LIN {X 0,Y 347.835,Z 893.328,A -85,B 0,C 180,E1 -23554.002,E2 -23554.002} C_VEL
LIN {X 0,Y 356.996,Z 872.801,A -85,B 0,C 180,E1 -23555.35,E2 -23555.35} C_VEL
LIN {X 0,Y 365.708,Z 850.209,A -85,B 0,C 180,E1 -23556.534,E2 -23556.534} C_VEL
LIN {X 0,Y 372.164,Z 830.904,A -85,B 0,C 180,E1 -23557.35,E2 -23557.35} C_VEL
LIN {X 0,Y 378.965,Z 806.777,A -85,B 0,C 180,E1 -23558.164,E2 -23558.164} C_VEL
LIN {X 0,Y 383.904,Z 784.469,A -85,B 0,C 180,E1 -23558.738,E2 -23558.738} C_VEL
LIN {X 0,Y 388.031,Z 759.695,A -85,B 0,C 180,E1 -23559.245,E2 -23559.245} C_VEL
LIN {X 0,Y 393.244,Z 706.009,A -85,B 0,C 180,E1 -23560.109,E2 -23560.109} C_VEL
LIN {X 0,Y 405.179,Z 577.067,A -85,B 0,C 180,E1 -23562.107,E2 -23562.107} C_VEL
LIN {X 0,Y 400.868,Z 567.631,A -85,B 0,C 180,E1 -23564.706,E2 -23564.706} C_VEL
LIN {X 0,Y 397.081,Z 560.851,A -85,B 0,C 180,E1 -23567.345,E2 -23567.345} C_VEL
LIN {X 0,Y 394.785,Z 556.79,A -85,B 0,C 180,E1 -23569.271,E2 -23569.271} C_VEL
LIN {X 0,Y 393.127,Z 553.806,A -85,B 0,C 180,E1 -23570.927,E2 -23570.927} C_VEL
LIN {X 0,Y 390.899,Z 549.726,A -85,B 0,C 180,E1 -23573.833,E2 -23573.833} C_VEL
LIN {X 0,Y 389.05,Z 545.081,A -85,B 0,C 180,E1 -23580.295,E2 -23580.295} C_VEL
LIN {X 0,Y 391.195,Z 550.264,A -85,B 0,C 180,E1 -23587.047,E2 -23587.047} C_VEL
LIN {X 0,Y 393.909,Z 555.208,A -85,B 0,C 180,E1 -23590.309,E2 -23590.309} C_VEL
LIN {X 0,Y 396.663,Z 560.048,A -85,B 0,C 180,E1 -23592.742,E2 -23592.742} C_VEL
LIN {X 0,Y 400.307,Z 566.598,A -85,B 0,C 180,E1 -23595.353,E2 -23595.353} C_VEL
LIN {X 0,Y 405.195,Z 575.818,A -85,B 0,C 180,E1 -23598.251,E2 -23598.251} C_VEL
LIN {X 0,Y 389.01,Z 748.36,A -85,B 0,C 180,E1 -23600.94,E2 -23600.94} C_VEL
LIN {X 0,Y 384.925,Z 774.814,A -85,B 0,C 180,E1 -23601.482,E2 -23601.482} C_VEL
LIN {X 0,Y 380.503,Z 795.662,A -85,B 0,C 180,E1 -23602.045,E2 -23602.045} C_VEL
LIN {X 0,Y 373.946,Z 820.335,A -85,B 0,C 180,E1 -23602.905,E2 -23602.905} C_VEL
LIN {X 0,Y 367.245,Z 840.974,A -85,B 0,C 180,E1 -23603.82,E2 -23603.82} C_VEL
LIN {X 0,Y 358.727,Z 863.66,A -85,B 0,C 180,E1 -23605.058,E2 -23605.058} C_VEL
LIN {X 0,Y 349.576,Z 884.374,A -85,B 0,C 180,E1 -23606.457,E2 -23606.457} C_VEL
LIN {X 0,Y 339.93,Z 904.027,A -85,B 0,C 180,E1 -23608.063,E2 -23608.063} C_VEL
LIN {X 0,Y 329.108,Z 923.521,A -85,B 0,C 180,E1 -23610.017,E2 -23610.017} C_VEL
LIN {X 0,Y 319.02,Z 940.165,A -85,B 0,C 180,E1 -23612.025,E2 -23612.025} C_VEL
LIN {X 0,Y 306.526,Z 958.98,A -85,B 0,C 180,E1 -23614.81,E2 -23614.81} C_VEL
LIN {X 0,Y 296.049,Z 973.609,A -85,B 0,C 180,E1 -23617.468,E2 -23617.468} C_VEL
LIN {X 0,Y 283.786,Z 989.665,A -85,B 0,C 180,E1 -23621.062,E2 -23621.062} C_VEL
LIN {X 0,Y 273.785,Z 1002.093,A -85,B 0,C 180,E1 -23624.524,E2 -23624.524} C_VEL
LIN {X 0,Y 263.22,Z 1014.833,A -85,B 0,C 180,E1 -23628.916,E2 -23628.916} C_VEL
LIN {X 0,Y 254.603,Z 1024.994,A -85,B 0,C 180,E1 -23633.349,E2 -23633.349} C_VEL
LIN {X 0,Y 246.801,Z 1034.427,A -85,B 0,C 180,E1 -23638.491,E2 -23638.491} C_VEL
LIN {X 0,Y 240.758,Z 1041.973,A -85,B 0,C 180,E1 -23643.882,E2 -23643.882} C_VEL
LIN {X 0,Y 236.318,Z 1048.28,A -85,B 0,C 180,E1 -23649.699,E2 -23649.699} C_VEL
LIN {X 0,Y 233.696,Z 1052.582,A -85,B 0,C 180,E1 -23655.378,E2 -23655.378} C_VEL
LIN {X 0,Y 232.543,Z 1055.206,A -85,B 0,C 180,E1 -23660.347,E2 -23660.347} C_VEL
LIN {X 0,Y 232.083,Z 1056.918,A -85,B 0,C 180,E1 -23665.8,E2 -23665.8} C_VEL
LIN {X 0,Y 232.025,Z 1057.239,A -85,B 0,C 180,E1 -23670.988,E2 -23670.988} C_VEL
LIN {X 0,Y 232.144,Z 1056.542,A -85,B 0,C 180,E1 -23675.751,E2 -23675.751} C_VEL
LIN {X 0,Y 232.638,Z 1054.939,A -85,B 0,C 180,E1 -23680.4,E2 -23680.4} C_VEL
LIN {X 0,Y 234.023,Z 1052.049,A -85,B 0,C 180,E1 -23685.615,E2 -23685.615} C_VEL
LIN {X 0,Y 237.201,Z 1046.942,A -85,B 0,C 180,E1 -23691.775,E2 -23691.775} C_VEL
LIN {X 0,Y 241.377,Z 1041.246,A -85,B 0,C 180,E1 -23696.842,E2 -23696.842} C_VEL
LIN {X 0,Y 248.254,Z 1032.711,A -85,B 0,C 180,E1 -23702.664,E2 -23702.664} C_VEL
LIN {X 0,Y 255.637,Z 1023.876,A -85,B 0,C 180,E1 -23707.32,E2 -23707.32} C_VEL
LIN {X 0,Y 265.345,Z 1012.444,A -85,B 0,C 180,E1 -23712.125,E2 -23712.125} C_VEL
LIN {X 0,Y 275.066,Z 1000.672,A -85,B 0,C 180,E1 -23716.034,E2 -23716.034} C_VEL
LIN {X 0,Y 285.965,Z 987.176,A -85,B 0,C 180,E1 -23719.694,E2 -23719.694} C_VEL
LIN {X 0,Y 297.122,Z 972.362,A -85,B 0,C 180,E1 -23722.898,E2 -23722.898} C_VEL
LIN {X 0,Y 307.93,Z 957.247,A -85,B 0,C 180,E1 -23725.597,E2 -23725.597} C_VEL
LIN {X 0,Y 319.887,Z 939.064,A -85,B 0,C 180,E1 -23728.234,E2 -23728.234} C_VEL
LIN {X 0,Y 330.019,Z 922.313,A -85,B 0,C 180,E1 -23730.231,E2 -23730.231} C_VEL
LIN {X 0,Y 341.605,Z 901.102,A -85,B 0,C 180,E1 -23732.305,E2 -23732.305} C_VEL
LIN {X 0,Y 350.412,Z 883.055,A -85,B 0,C 180,E1 -23733.75,E2 -23733.75} C_VEL
LIN {X 0,Y 359.976,Z 861.087,A -85,B 0,C 180,E1 -23735.201,E2 -23735.201} C_VEL
LIN {X 0,Y 367.879,Z 839.801,A -85,B 0,C 180,E1 -23736.343,E2 -23736.343} C_VEL
LIN {X 0,Y 375.388,Z 816.305,A -85,B 0,C 180,E1 -23737.361,E2 -23737.361} C_VEL
LIN {X 0,Y 381.309,Z 793.174,A -85,B 0,C 180,E1 -23738.135,E2 -23738.135} C_VEL
LIN {X 0,Y 386.229,Z 769.254,A -85,B 0,C 180,E1 -23738.756,E2 -23738.756} C_VEL
LIN {X 0,Y 389.656,Z 744.741,A -85,B 0,C 180,E1 -23739.225,E2 -23739.225} C_VEL
LIN {X 0,Y 405.413,Z 575.97,A -85,B 0,C 180,E1 -23741.857,E2 -23741.857} C_VEL
LIN {X 0,Y 400.628,Z 566.958,A -85,B 0,C 180,E1 -23744.696,E2 -23744.696} C_VEL
LIN {X 0,Y 397.121,Z 560.633,A -85,B 0,C 180,E1 -23747.199,E2 -23747.199} C_VEL
LIN {X 0,Y 395.089,Z 557.156,A -85,B 0,C 180,E1 -23748.911,E2 -23748.911} C_VEL
LIN {X 0,Y 393.763,Z 554.568,A -85,B 0,C 180,E1 -23750.233,E2 -23750.233} C_VEL
LIN {X 0,Y 392.838,Z 553.605,A -85,B 0,C 180,E1 -23751.18,E2 -23751.18} C_VEL
LIN {X 0,Y 391.337,Z 554.58,A -85,B 0,C 180,E1 -23752.628,E2 -23752.628} C_VEL
LIN {X 0,Y 389.554,Z 556.788,A -85,B 0,C 180,E1 -23754.674,E2 -23754.674} C_VEL
LIN {X 0,Y 389.136,Z 556.727,A -85,B 0,C 180,E1 -23755.421,E2 -23755.421} C_VEL
LIN {X 0,Y 388.33,Z 553.902,A -85,B 0,C 180,E1 -23760,E2 -23760} C_VEL
LIN {X 0,Y 390.299,Z 558.224,A -85,B 0,C 180,E1 -23766.325,E2 -23766.325} C_VEL
LIN {X 0,Y 392.89,Z 563.078,A -85,B 0,C 180,E1 -23769.596,E2 -23769.596} C_VEL
LIN {X 0,Y 395.281,Z 567.502,A -85,B 0,C 180,E1 -23771.823,E2 -23771.823} C_VEL
LIN {X 0,Y 398.829,Z 573.955,A -85,B 0,C 180,E1 -23774.482,E2 -23774.482} C_VEL
LIN {X 0,Y 401.266,Z 579.253,A -85,B 0,C 180,E1 -23776.094,E2 -23776.094} C_VEL
LIN {X 0,Y 402.503,Z 582.459,A -85,B 0,C 180,E1 -23776.88,E2 -23776.88} C_VEL
LIN {X 0,Y 385.936,Z 755.658,A -85,B 0,C 180,E1 -23779.56,E2 -23779.56} C_VEL
LIN {X 0,Y 381.709,Z 782.23,A -85,B 0,C 180,E1 -23780.078,E2 -23780.078} C_VEL
LIN {X 0,Y 376.982,Z 803.644,A -85,B 0,C 180,E1 -23780.604,E2 -23780.604} C_VEL
LIN {X 0,Y 369.986,Z 828.756,A -85,B 0,C 180,E1 -23781.406,E2 -23781.406} C_VEL
LIN {X 0,Y 363.401,Z 848.284,A -85,B 0,C 180,E1 -23782.199,E2 -23782.199} C_VEL
LIN {X 0,Y 354.645,Z 870.927,A -85,B 0,C 180,E1 -23783.34,E2 -23783.34} C_VEL
LIN {X 0,Y 345.022,Z 892.161,A -85,B 0,C 180,E1 -23784.696,E2 -23784.696} C_VEL
LIN {X 0,Y 334.593,Z 912.794,A -85,B 0,C 180,E1 -23786.296,E2 -23786.296} C_VEL
LIN {X 0,Y 323.349,Z 932.438,A -85,B 0,C 180,E1 -23788.2,E2 -23788.2} C_VEL
LIN {X 0,Y 312.514,Z 949.839,A -85,B 0,C 180,E1 -23790.246,E2 -23790.246} C_VEL
LIN {X 0,Y 300.014,Z 968.143,A -85,B 0,C 180,E1 -23792.905,E2 -23792.905} C_VEL
LIN {X 0,Y 288.971,Z 983.211,A -85,B 0,C 180,E1 -23795.596,E2 -23795.596} C_VEL
LIN {X 0,Y 276.215,Z 999.555,A -85,B 0,C 180,E1 -23799.224,E2 -23799.224} C_VEL
LIN {X 0,Y 265.688,Z 1012.399,A -85,B 0,C 180,E1 -23802.789,E2 -23802.789} C_VEL
LIN {X 0,Y 253.914,Z 1026.348,A -85,B 0,C 180,E1 -23807.671,E2 -23807.671} C_VEL
LIN {X 0,Y 245.528,Z 1036.235,A -85,B 0,C 180,E1 -23812.053,E2 -23812.053} C_VEL
LIN {X 0,Y 236.986,Z 1046.589,A -85,B 0,C 180,E1 -23817.885,E2 -23817.885} C_VEL
LIN {X 0,Y 231.559,Z 1053.665,A -85,B 0,C 180,E1 -23823.038,E2 -23823.038} C_VEL
LIN {X 0,Y 227.283,Z 1060.146,A -85,B 0,C 180,E1 -23829.124,E2 -23829.124} C_VEL
LIN {X 0,Y 225.031,Z 1064.472,A -85,B 0,C 180,E1 -23834.802,E2 -23834.802} C_VEL
LIN {X 0,Y 224.137,Z 1067.258,A -85,B 0,C 180,E1 -23839.98,E2 -23839.98} C_VEL
LIN {X 0,Y 223.98,Z 1069.011,A -85,B 0,C 180,E1 -23845.391,E2 -23845.391} C_VEL
LIN {X 0,Y 224.019,Z 1069.447,A -85,B 0,C 180,E1 -23850.511,E2 -23850.511} C_VEL
LIN {X 0,Y 223.982,Z 1068.773,A -85,B 0,C 180,E1 -23855.43,E2 -23855.43} C_VEL
LIN {X 0,Y 224.163,Z 1067.118,A -85,B 0,C 180,E1 -23860.278,E2 -23860.278} C_VEL
LIN {X 0,Y 225.102,Z 1064.276,A -85,B 0,C 180,E1 -23865.457,E2 -23865.457} C_VEL
LIN {X 0,Y 227.71,Z 1059.396,A -85,B 0,C 180,E1 -23871.644,E2 -23871.644} C_VEL
LIN {X 0,Y 232.007,Z 1052.984,A -85,B 0,C 180,E1 -23877.461,E2 -23877.461} C_VEL
LIN {X 0,Y 238.204,Z 1045.073,A -85,B 0,C 180,E1 -23883.072,E2 -23883.072} C_VEL
LIN {X 0,Y 246.352,Z 1035.142,A -85,B 0,C 180,E1 -23888.432,E2 -23888.432} C_VEL
LIN {X 0,Y 255.749,Z 1024.154,A -85,B 0,C 180,E1 -23893.172,E2 -23893.172} C_VEL
LIN {X 0,Y 266.497,Z 1011.26,A -85,B 0,C 180,E1 -23897.518,E2 -23897.518} C_VEL
LIN {X 0,Y 277.466,Z 997.863,A -85,B 0,C 180,E1 -23901.168,E2 -23901.168} C_VEL
LIN {X 0,Y 289.588,Z 982.165,A -85,B 0,C 180,E1 -23904.573,E2 -23904.573} C_VEL
LIN {X 0,Y 300.731,Z 966.912,A -85,B 0,C 180,E1 -23907.266,E2 -23907.266} C_VEL
LIN {X 0,Y 313.412,Z 948.132,A -85,B 0,C 180,E1 -23909.941,E2 -23909.941} C_VEL
LIN {X 0,Y 323.697,Z 931.53,A -85,B 0,C 180,E1 -23911.872,E2 -23911.872} C_VEL
LIN {X 0,Y 335.331,Z 910.95,A -85,B 0,C 180,E1 -23913.834,E2 -23913.834} C_VEL
LIN {X 0,Y 344.999,Z 891.755,A -85,B 0,C 180,E1 -23915.312,E2 -23915.312} C_VEL
LIN {X 0,Y 354.893,Z 869.78,A -85,B 0,C 180,E1 -23916.705,E2 -23916.705} C_VEL
LIN {X 0,Y 363.376,Z 847.717,A -85,B 0,C 180,E1 -23917.81,E2 -23917.81} C_VEL
LIN {X 0,Y 370.996,Z 824.871,A -85,B 0,C 180,E1 -23918.724,E2 -23918.724} C_VEL
LIN {X 0,Y 377.303,Z 801.317,A -85,B 0,C 180,E1 -23919.444,E2 -23919.444} C_VEL
LIN {X 0,Y 382.253,Z 778.324,A -85,B 0,C 180,E1 -23919.995,E2 -23919.995} C_VEL
LIN {X 0,Y 385.966,Z 753.258,A -85,B 0,C 180,E1 -23920.467,E2 -23920.467} C_VEL
LIN {X 0,Y 402.254,Z 581.98,A -85,B 0,C 180,E1 -23923.133,E2 -23923.133} C_VEL
LIN {X 0,Y 399.045,Z 574.683,A -85,B 0,C 180,E1 -23925.192,E2 -23925.192} C_VEL
LIN {X 0,Y 395.538,Z 568.236,A -85,B 0,C 180,E1 -23927.74,E2 -23927.74} C_VEL
LIN {X 0,Y 393.361,Z 564.263,A -85,B 0,C 180,E1 -23929.646,E2 -23929.646} C_VEL
LIN {X 0,Y 391.874,Z 561.512,A -85,B 0,C 180,E1 -23931.194,E2 -23931.194} C_VEL
LIN {X 0,Y 389.826,Z 557.61,A -85,B 0,C 180,E1 -23933.963,E2 -23933.963} C_VEL
LIN {X 0,Y 388.07,Z 553.065,A -85,B 0,C 180,E1 -23940.295,E2 -23940.295} C_VEL
LIN {X 0,Y 390.11,Z 558.197,A -85,B 0,C 180,E1 -23946.919,E2 -23946.919} C_VEL
LIN {X 0,Y 392.633,Z 562.902,A -85,B 0,C 180,E1 -23950.046,E2 -23950.046} C_VEL
LIN {X 0,Y 395.301,Z 567.74,A -85,B 0,C 180,E1 -23952.483,E2 -23952.483} C_VEL
LIN {X 0,Y 398.867,Z 574.383,A -85,B 0,C 180,E1 -23955.112,E2 -23955.112} C_VEL
LIN {X 0,Y 402.28,Z 581.103,A -85,B 0,C 180,E1 -23957.247,E2 -23957.247} C_VEL
LIN {X 0,Y 386.223,Z 748.596,A -85,B 0,C 180,E1 -23959.831,E2 -23959.831} C_VEL
LIN {X 0,Y 382.065,Z 775.041,A -85,B 0,C 180,E1 -23960.365,E2 -23960.365} C_VEL
LIN {X 0,Y 377.539,Z 796.006,A -85,B 0,C 180,E1 -23960.92,E2 -23960.92} C_VEL
LIN {X 0,Y 370.894,Z 820.557,A -85,B 0,C 180,E1 -23961.762,E2 -23961.762} C_VEL
LIN {X 0,Y 364.072,Z 841.195,A -85,B 0,C 180,E1 -23962.663,E2 -23962.663} C_VEL
LIN {X 0,Y 355.785,Z 862.969,A -85,B 0,C 180,E1 -23963.826,E2 -23963.826} C_VEL
LIN {X 0,Y 346.372,Z 883.931,A -85,B 0,C 180,E1 -23965.212,E2 -23965.212} C_VEL
LIN {X 0,Y 337.315,Z 902.058,A -85,B 0,C 180,E1 -23966.655,E2 -23966.655} C_VEL
LIN {X 0,Y 325.851,Z 922.533,A -85,B 0,C 180,E1 -23968.646,E2 -23968.646} C_VEL
LIN {X 0,Y 315.826,Z 938.734,A -85,B 0,C 180,E1 -23970.556,E2 -23970.556} C_VEL
LIN {X 0,Y 303.797,Z 956.658,A -85,B 0,C 180,E1 -23973.118,E2 -23973.118} C_VEL
LIN {X 0,Y 292.406,Z 972.156,A -85,B 0,C 180,E1 -23975.863,E2 -23975.863} C_VEL
LIN {X 0,Y 280.816,Z 987.093,A -85,B 0,C 180,E1 -23979.084,E2 -23979.084} C_VEL
LIN {X 0,Y 269.51,Z 1000.635,A -85,B 0,C 180,E1 -23982.761,E2 -23982.761} C_VEL
LIN {X 0,Y 259.43,Z 1012.375,A -85,B 0,C 180,E1 -23986.683,E2 -23986.683} C_VEL
LIN {X 0,Y 249.261,Z 1023.861,A -85,B 0,C 180,E1 -23991.555,E2 -23991.555} C_VEL
LIN {X 0,Y 241.36,Z 1032.85,A -85,B 0,C 180,E1 -23996.377,E2 -23996.377} C_VEL
LIN {X 0,Y 234.159,Z 1041.303,A -85,B 0,C 180,E1 -24002.261,E2 -24002.261} C_VEL
LIN {X 0,Y 229.684,Z 1047.025,A -85,B 0,C 180,E1 -24007.475,E2 -24007.475} C_VEL
LIN {X 0,Y 226.24,Z 1052.18,A -85,B 0,C 180,E1 -24013.833,E2 -24013.833} C_VEL
LIN {X 0,Y 224.717,Z 1055.093,A -85,B 0,C 180,E1 -24019.229,E2 -24019.229} C_VEL
LIN {X 0,Y 224.158,Z 1056.737,A -85,B 0,C 180,E1 -24024.115,E2 -24024.115} C_VEL
LIN {X 0,Y 224.027,Z 1057.44,A -85,B 0,C 180,E1 -24028.977,E2 -24028.977} C_VEL
LIN {X 0,Y 224.09,Z 1057.164,A -85,B 0,C 180,E1 -24034.351,E2 -24034.351} C_VEL
LIN {X 0,Y 224.582,Z 1055.484,A -85,B 0,C 180,E1 -24040,E2 -24040} C_VEL
LIN {X 0,Y 225.839,Z 1052.874,A -85,B 0,C 180,E1 -24045.162,E2 -24045.162} C_VEL
LIN {X 0,Y 228.796,Z 1048.397,A -85,B 0,C 180,E1 -24051.268,E2 -24051.268} C_VEL
LIN {X 0,Y 233.361,Z 1042.353,A -85,B 0,C 180,E1 -24057.013,E2 -24057.013} C_VEL
LIN {X 0,Y 239.429,Z 1035.18,A -85,B 0,C 180,E1 -24062.313,E2 -24062.313} C_VEL
LIN {X 0,Y 247.945,Z 1025.449,A -85,B 0,C 180,E1 -24067.805,E2 -24067.805} C_VEL
LIN {X 0,Y 256.495,Z 1015.819,A -85,B 0,C 180,E1 -24072.106,E2 -24072.106} C_VEL
LIN {X 0,Y 267.838,Z 1002.771,A -85,B 0,C 180,E1 -24076.717,E2 -24076.717} C_VEL
LIN {X 0,Y 278.342,Z 990.221,A -85,B 0,C 180,E1 -24080.25,E2 -24080.25} C_VEL
LIN {X 0,Y 291,Z 974.252,A -85,B 0,C 180,E1 -24083.85,E2 -24083.85} C_VEL
LIN {X 0,Y 301.322,Z 960.303,A -85,B 0,C 180,E1 -24086.398,E2 -24086.398} C_VEL
LIN {X 0,Y 313.583,Z 942.582,A -85,B 0,C 180,E1 -24089.063,E2 -24089.063} C_VEL
LIN {X 0,Y 324.607,Z 924.941,A -85,B 0,C 180,E1 -24091.205,E2 -24091.205} C_VEL
LIN {X 0,Y 335.672,Z 905.662,A -85,B 0,C 180,E1 -24093.144,E2 -24093.144} C_VEL
LIN {X 0,Y 345.903,Z 885.378,A -85,B 0,C 180,E1 -24094.794,E2 -24094.794} C_VEL
LIN {X 0,Y 355.023,Z 865.225,A -85,B 0,C 180,E1 -24096.143,E2 -24096.143} C_VEL
LIN {X 0,Y 363.927,Z 842.261,A -85,B 0,C 180,E1 -24097.393,E2 -24097.393} C_VEL
LIN {X 0,Y 370.753,Z 821.765,A -85,B 0,C 180,E1 -24098.293,E2 -24098.293} C_VEL
LIN {X 0,Y 377.704,Z 796.339,A -85,B 0,C 180,E1 -24099.173,E2 -24099.173} C_VEL
LIN {X 0,Y 382.228,Z 775.446,A -85,B 0,C 180,E1 -24099.729,E2 -24099.729} C_VEL
LIN {X 0,Y 386.349,Z 749.637,A -85,B 0,C 180,E1 -24100.255,E2 -24100.255} C_VEL
LIN {X 0,Y 395.791,Z 651.868,A -85,B 0,C 180,E1 -24101.779,E2 -24101.779} C_VEL
LIN {X 0,Y 402.488,Z 581.077,A -85,B 0,C 180,E1 -24102.879,E2 -24102.879} C_VEL
LIN {X 0,Y 398.217,Z 572.864,A -85,B 0,C 180,E1 -24105.606,E2 -24105.606} C_VEL
LIN {X 0,Y 394.679,Z 566.202,A -85,B 0,C 180,E1 -24108.381,E2 -24108.381} C_VEL
LIN {X 0,Y 391.99,Z 561.546,A -85,B 0,C 180,E1 -24111.048,E2 -24111.048} C_VEL
LIN {X 0,Y 390.009,Z 557.709,A -85,B 0,C 180,E1 -24113.818,E2 -24113.818} C_VEL
LIN {X 0,Y 389.136,Z 556.727,A -85,B 0,C 180,E1 -24115.421,E2 -24115.421} C_VEL
LIN {X 0,Y 388.526,Z 556.957,A -85,B 0,C 180,E1 -24116.725,E2 -24116.725} C_VEL
LIN {X 0,Y 387.342,Z 562.179,A -85,B 0,C 180,E1 -24120.541,E2 -24120.541} C_VEL
LIN {X 0,Y 387.342,Z 562.238,A -85,B 0,C 180,E1 -24120.624,E2 -24120.624} C_VEL
LIN {X 0,Y 389.22,Z 566.147,A -85,B 0,C 180,E1 -24126.194,E2 -24126.194} C_VEL
LIN {X 0,Y 391.624,Z 570.769,A -85,B 0,C 180,E1 -24129.33,E2 -24129.33} C_VEL
LIN {X 0,Y 393.943,Z 575.21,A -85,B 0,C 180,E1 -24131.567,E2 -24131.567} C_VEL
LIN {X 0,Y 397.303,Z 581.526,A -85,B 0,C 180,E1 -24134.167,E2 -24134.167} C_VEL
LIN {X 0,Y 399.766,Z 587.148,A -85,B 0,C 180,E1 -24135.852,E2 -24135.852} C_VEL
LIN {X 0,Y 383.322,Z 755.464,A -85,B 0,C 180,E1 -24138.429,E2 -24138.429} C_VEL
LIN {X 0,Y 379.026,Z 782.029,A -85,B 0,C 180,E1 -24138.937,E2 -24138.937} C_VEL
LIN {X 0,Y 374.227,Z 803.44,A -85,B 0,C 180,E1 -24139.451,E2 -24139.451} C_VEL
LIN {X 0,Y 367.087,Z 828.651,A -85,B 0,C 180,E1 -24140.239,E2 -24140.239} C_VEL
LIN {X 0,Y 360.013,Z 849.21,A -85,B 0,C 180,E1 -24141.061,E2 -24141.061} C_VEL
LIN {X 0,Y 350.975,Z 871.908,A -85,B 0,C 180,E1 -24142.197,E2 -24142.197} C_VEL
LIN {X 0,Y 341.309,Z 892.765,A -85,B 0,C 180,E1 -24143.515,E2 -24143.515} C_VEL
LIN {X 0,Y 330.675,Z 913.297,A -85,B 0,C 180,E1 -24145.092,E2 -24145.092} C_VEL
LIN {X 0,Y 319.19,Z 932.836,A -85,B 0,C 180,E1 -24146.973,E2 -24146.973} C_VEL
LIN {X 0,Y 307.378,Z 951.301,A -85,B 0,C 180,E1 -24149.141,E2 -24149.141} C_VEL
LIN {X 0,Y 294.996,Z 968.776,A -85,B 0,C 180,E1 -24151.705,E2 -24151.705} C_VEL
LIN {X 0,Y 283.598,Z 983.847,A -85,B 0,C 180,E1 -24154.409,E2 -24154.409} C_VEL
LIN {X 0,Y 271.059,Z 999.336,A -85,B 0,C 180,E1 -24157.869,E2 -24157.869} C_VEL
LIN {X 0,Y 260.126,Z 1012.18,A -85,B 0,C 180,E1 -24161.448,E2 -24161.448} C_VEL
LIN {X 0,Y 247.845,Z 1026.128,A -85,B 0,C 180,E1 -24166.38,E2 -24166.38} C_VEL
LIN {X 0,Y 239.039,Z 1036.015,A -85,B 0,C 180,E1 -24170.83,E2 -24170.83} C_VEL
LIN {X 0,Y 230.013,Z 1046.369,A -85,B 0,C 180,E1 -24176.788,E2 -24176.788} C_VEL
LIN {X 0,Y 224.23,Z 1053.446,A -85,B 0,C 180,E1 -24182.081,E2 -24182.081} C_VEL
LIN {X 0,Y 219.627,Z 1059.927,A -85,B 0,C 180,E1 -24188.36,E2 -24188.36} C_VEL
LIN {X 0,Y 217.168,Z 1064.255,A -85,B 0,C 180,E1 -24194.237,E2 -24194.237} C_VEL
LIN {X 0,Y 216.172,Z 1067.042,A -85,B 0,C 180,E1 -24199.607,E2 -24199.607} C_VEL
LIN {X 0,Y 215.982,Z 1068.797,A -85,B 0,C 180,E1 -24205.22,E2 -24205.22} C_VEL
LIN {X 0,Y 216.024,Z 1069.256,A -85,B 0,C 180,E1 -24210.265,E2 -24210.265} C_VEL
LIN {X 0,Y 215.984,Z 1068.585,A -85,B 0,C 180,E1 -24215.532,E2 -24215.532} C_VEL
LIN {X 0,Y 216.199,Z 1066.902,A -85,B 0,C 180,E1 -24220.661,E2 -24220.661} C_VEL
LIN {X 0,Y 217.247,Z 1064.058,A -85,B 0,C 180,E1 -24226.03,E2 -24226.03} C_VEL
LIN {X 0,Y 220.088,Z 1059.176,A -85,B 0,C 180,E1 -24232.434,E2 -24232.434} C_VEL
LIN {X 0,Y 224.708,Z 1052.763,A -85,B 0,C 180,E1 -24238.432,E2 -24238.432} C_VEL
LIN {X 0,Y 231.308,Z 1044.85,A -85,B 0,C 180,E1 -24244.191,E2 -24244.191} C_VEL
LIN {X 0,Y 239.846,Z 1034.987,A -85,B 0,C 180,E1 -24249.631,E2 -24249.631} C_VEL
LIN {X 0,Y 249.763,Z 1023.931,A -85,B 0,C 180,E1 -24254.474,E2 -24254.474} C_VEL
LIN {X 0,Y 260.66,Z 1011.398,A -85,B 0,C 180,E1 -24258.751,E2 -24258.751} C_VEL
LIN {X 0,Y 271.815,Z 998.273,A -85,B 0,C 180,E1 -24262.364,E2 -24262.364} C_VEL
LIN {X 0,Y 284.232,Z 982.796,A -85,B 0,C 180,E1 -24265.761,E2 -24265.761} C_VEL
LIN {X 0,Y 295.01,Z 968.512,A -85,B 0,C 180,E1 -24268.308,E2 -24268.308} C_VEL
LIN {X 0,Y 307.72,Z 950.474,A -85,B 0,C 180,E1 -24270.935,E2 -24270.935} C_VEL
LIN {X 0,Y 319.168,Z 932.533,A -85,B 0,C 180,E1 -24273.034,E2 -24273.034} C_VEL
LIN {X 0,Y 330.653,Z 912.94,A -85,B 0,C 180,E1 -24274.915,E2 -24274.915} C_VEL
LIN {X 0,Y 341.285,Z 892.349,A -85,B 0,C 180,E1 -24276.494,E2 -24276.494} C_VEL
LIN {X 0,Y 350.952,Z 871.453,A -85,B 0,C 180,E1 -24277.812,E2 -24277.812} C_VEL
LIN {X 0,Y 359.988,Z 848.629,A -85,B 0,C 180,E1 -24278.949,E2 -24278.949} C_VEL
LIN {X 0,Y 367.517,Z 826.592,A -85,B 0,C 180,E1 -24279.822,E2 -24279.822} C_VEL
LIN {X 0,Y 374.231,Z 802.425,A -85,B 0,C 180,E1 -24280.561,E2 -24280.561} C_VEL
LIN {X 0,Y 379.017,Z 780.857,A -85,B 0,C 180,E1 -24281.074,E2 -24281.074} C_VEL
LIN {X 0,Y 383.196,Z 754.379,A -85,B 0,C 180,E1 -24281.576,E2 -24281.576} C_VEL
LIN {X 0,Y 399.508,Z 586.924,A -85,B 0,C 180,E1 -24284.148,E2 -24284.148} C_VEL
LIN {X 0,Y 397.002,Z 581.207,A -85,B 0,C 180,E1 -24285.859,E2 -24285.859} C_VEL
LIN {X 0,Y 392.968,Z 573.447,A -85,B 0,C 180,E1 -24289.073,E2 -24289.073} C_VEL
LIN {X 0,Y 390.63,Z 569.218,A -85,B 0,C 180,E1 -24291.462,E2 -24291.462} C_VEL
LIN {X 0,Y 388.661,Z 565.407,A -85,B 0,C 180,E1 -24294.242,E2 -24294.242} C_VEL
LIN {X 0,Y 387.09,Z 561.048,A -85,B 0,C 180,E1 -24300.296,E2 -24300.296} C_VEL
LIN {X 0,Y 388.986,Z 566.008,A -85,B 0,C 180,E1 -24306.717,E2 -24306.717} C_VEL
LIN {X 0,Y 391.365,Z 570.596,A -85,B 0,C 180,E1 -24309.782,E2 -24309.782} C_VEL
LIN {X 0,Y 393.964,Z 575.461,A -85,B 0,C 180,E1 -24312.235,E2 -24312.235} C_VEL
LIN {X 0,Y 397.588,Z 582.47,A -85,B 0,C 180,E1 -24314.976,E2 -24314.976} C_VEL
LIN {X 0,Y 399.474,Z 586.526,A -85,B 0,C 180,E1 -24316.23,E2 -24316.23} C_VEL
LIN {X 0,Y 383.559,Z 749.024,A -85,B 0,C 180,E1 -24318.71,E2 -24318.71} C_VEL
LIN {X 0,Y 379.331,Z 775.378,A -85,B 0,C 180,E1 -24319.234,E2 -24319.234} C_VEL
LIN {X 0,Y 374.723,Z 796.351,A -85,B 0,C 180,E1 -24319.779,E2 -24319.779} C_VEL
LIN {X 0,Y 367.993,Z 820.78,A -85,B 0,C 180,E1 -24320.601,E2 -24320.601} C_VEL
LIN {X 0,Y 361.05,Z 841.417,A -85,B 0,C 180,E1 -24321.485,E2 -24321.485} C_VEL
LIN {X 0,Y 352.476,Z 863.496,A -85,B 0,C 180,E1 -24322.646,E2 -24322.646} C_VEL
LIN {X 0,Y 342.687,Z 884.816,A -85,B 0,C 180,E1 -24324.039,E2 -24324.039} C_VEL
LIN {X 0,Y 332.617,Z 904.469,A -85,B 0,C 180,E1 -24325.6,E2 -24325.6} C_VEL
LIN {X 0,Y 321.293,Z 923.962,A -85,B 0,C 180,E1 -24327.509,E2 -24327.509} C_VEL
LIN {X 0,Y 311.049,Z 940.057,A -85,B 0,C 180,E1 -24329.408,E2 -24329.408} C_VEL
LIN {X 0,Y 297.716,Z 959.149,A -85,B 0,C 180,E1 -24332.183,E2 -24332.183} C_VEL
LIN {X 0,Y 287.041,Z 973.214,A -85,B 0,C 180,E1 -24334.705,E2 -24334.705} C_VEL
LIN {X 0,Y 274.506,Z 988.721,A -85,B 0,C 180,E1 -24338.115,E2 -24338.115} C_VEL
LIN {X 0,Y 263.508,Z 1001.419,A -85,B 0,C 180,E1 -24341.624,E2 -24341.624} C_VEL
LIN {X 0,Y 252.527,Z 1013.727,A -85,B 0,C 180,E1 -24345.823,E2 -24345.823} C_VEL
LIN {X 0,Y 242.451,Z 1024.533,A -85,B 0,C 180,E1 -24350.572,E2 -24350.572} C_VEL
LIN {X 0,Y 233.983,Z 1033.733,A -85,B 0,C 180,E1 -24355.662,E2 -24355.662} C_VEL
LIN {X 0,Y 226.67,Z 1041.82,A -85,B 0,C 180,E1 -24361.549,E2 -24361.549} C_VEL
LIN {X 0,Y 221.785,Z 1047.741,A -85,B 0,C 180,E1 -24367.188,E2 -24367.188} C_VEL
LIN {X 0,Y 218.236,Z 1052.707,A -85,B 0,C 180,E1 -24373.771,E2 -24373.771} C_VEL
LIN {X 0,Y 216.74,Z 1055.418,A -85,B 0,C 180,E1 -24379.097,E2 -24379.097} C_VEL
LIN {X 0,Y 216.159,Z 1057.016,A -85,B 0,C 180,E1 -24384.159,E2 -24384.159} C_VEL
LIN {X 0,Y 216.026,Z 1057.698,A -85,B 0,C 180,E1 -24389.47,E2 -24389.47} C_VEL
LIN {X 0,Y 216.119,Z 1057.25,A -85,B 0,C 180,E1 -24395.043,E2 -24395.043} C_VEL
LIN {X 0,Y 216.678,Z 1055.589,A -85,B 0,C 180,E1 -24400.637,E2 -24400.637} C_VEL
LIN {X 0,Y 218.106,Z 1052.946,A -85,B 0,C 180,E1 -24405.966,E2 -24405.966} C_VEL
LIN {X 0,Y 221.379,Z 1048.37,A -85,B 0,C 180,E1 -24412.297,E2 -24412.297} C_VEL
LIN {X 0,Y 226.34,Z 1042.275,A -85,B 0,C 180,E1 -24418.209,E2 -24418.209} C_VEL
LIN {X 0,Y 233.203,Z 1034.705,A -85,B 0,C 180,E1 -24423.876,E2 -24423.876} C_VEL
LIN {X 0,Y 241.918,Z 1025.215,A -85,B 0,C 180,E1 -24429.226,E2 -24429.226} C_VEL
LIN {X 0,Y 251.911,Z 1014.515,A -85,B 0,C 180,E1 -24433.997,E2 -24433.997} C_VEL
LIN {X 0,Y 263.083,Z 1002.063,A -85,B 0,C 180,E1 -24438.308,E2 -24438.308} C_VEL
LIN {X 0,Y 274.364,Z 989.069,A -85,B 0,C 180,E1 -24441.924,E2 -24441.924} C_VEL
LIN {X 0,Y 286.897,Z 973.63,A -85,B 0,C 180,E1 -24445.336,E2 -24445.336} C_VEL
LIN {X 0,Y 297.568,Z 959.6,A -85,B 0,C 180,E1 -24447.863,E2 -24447.863} C_VEL
LIN {X 0,Y 310.545,Z 941.144,A -85,B 0,C 180,E1 -24450.57,E2 -24450.57} C_VEL
LIN {X 0,Y 321.369,Z 924.187,A -85,B 0,C 180,E1 -24452.582,E2 -24452.582} C_VEL
LIN {X 0,Y 332.855,Z 904.447,A -85,B 0,C 180,E1 -24454.515,E2 -24454.515} C_VEL
LIN {X 0,Y 342.542,Z 885.589,A -85,B 0,C 180,E1 -24456.016,E2 -24456.016} C_VEL
LIN {X 0,Y 351.695,Z 865.757,A -85,B 0,C 180,E1 -24457.325,E2 -24457.325} C_VEL
LIN {X 0,Y 360.58,Z 843.387,A -85,B 0,C 180,E1 -24458.528,E2 -24458.528} C_VEL
LIN {X 0,Y 367.448,Z 823.252,A -85,B 0,C 180,E1 -24459.404,E2 -24459.404} C_VEL
LIN {X 0,Y 374.39,Z 798.814,A -85,B 0,C 180,E1 -24460.25,E2 -24460.25} C_VEL
LIN {X 0,Y 379.189,Z 777.337,A -85,B 0,C 180,E1 -24460.824,E2 -24460.824} C_VEL
LIN {X 0,Y 383.356,Z 752.93,A -85,B 0,C 180,E1 -24461.328,E2 -24461.328} C_VEL
LIN {X 0,Y 388.692,Z 700.563,A -85,B 0,C 180,E1 -24462.149,E2 -24462.149} C_VEL
LIN {X 0,Y 399.734,Z 586.426,A -85,B 0,C 180,E1 -24463.88,E2 -24463.88} C_VEL
LIN {X 0,Y 395.755,Z 578.597,A -85,B 0,C 180,E1 -24466.633,E2 -24466.633} C_VEL
LIN {X 0,Y 392.799,Z 573.044,A -85,B 0,C 180,E1 -24469.142,E2 -24469.142} C_VEL
LIN {X 0,Y 390.881,Z 569.436,A -85,B 0,C 180,E1 -24471.171,E2 -24471.171} C_VEL
LIN {X 0,Y 388.853,Z 565.503,A -85,B 0,C 180,E1 -24474.096,E2 -24474.096} C_VEL
LIN {X 0,Y 387.353,Z 561.858,A -85,B 0,C 180,E1 -24480,E2 -24480} C_VEL
LIN {X 0,Y 387.342,Z 562.238,A -85,B 0,C 180,E1 -24480.624,E2 -24480.624} C_VEL
LIN {X 0,Y 387.305,Z 563.992,A -85,B 0,C 180,E1 -24481.743,E2 -24481.743} C_VEL
LIN {X 0,Y 387.45,Z 572.167,A -85,B 0,C 180,E1 -24484.643,E2 -24484.643} C_VEL
LIN {X 0,Y 387.889,Z 573.488,A -85,B 0,C 180,E1 -24485.604,E2 -24485.604} C_VEL
LIN {X 0,Y 390.367,Z 578.459,A -85,B 0,C 180,E1 -24489.063,E2 -24489.063} C_VEL
LIN {X 0,Y 392.702,Z 583.09,A -85,B 0,C 180,E1 -24491.388,E2 -24491.388} C_VEL
LIN {X 0,Y 395.886,Z 589.303,A -85,B 0,C 180,E1 -24493.92,E2 -24493.92} C_VEL
LIN {X 0,Y 397.105,Z 592.406,A -85,B 0,C 180,E1 -24494.819,E2 -24494.819} C_VEL
LIN {X 0,Y 380.859,Z 755.271,A -85,B 0,C 180,E1 -24497.283,E2 -24497.283} C_VEL
LIN {X 0,Y 376.49,Z 781.862,A -85,B 0,C 180,E1 -24497.782,E2 -24497.782} C_VEL
LIN {X 0,Y 371.6,Z 803.345,A -85,B 0,C 180,E1 -24498.285,E2 -24498.285} C_VEL
LIN {X 0,Y 364.41,Z 828.344,A -85,B 0,C 180,E1 -24499.046,E2 -24499.046} C_VEL
LIN {X 0,Y 357.188,Z 849.001,A -85,B 0,C 180,E1 -24499.851,E2 -24499.851} C_VEL
LIN {X 0,Y 347.996,Z 871.698,A -85,B 0,C 180,E1 -24500.962,E2 -24500.962} C_VEL
LIN {X 0,Y 338.151,Z 892.553,A -85,B 0,C 180,E1 -24502.253,E2 -24502.253} C_VEL
LIN {X 0,Y 327.304,Z 913.083,A -85,B 0,C 180,E1 -24503.801,E2 -24503.801} C_VEL
LIN {X 0,Y 315.567,Z 932.621,A -85,B 0,C 180,E1 -24505.65,E2 -24505.65} C_VEL
LIN {X 0,Y 303.643,Z 950.828,A -85,B 0,C 180,E1 -24507.758,E2 -24507.758} C_VEL
LIN {X 0,Y 290.758,Z 968.559,A -85,B 0,C 180,E1 -24510.326,E2 -24510.326} C_VEL
LIN {X 0,Y 279.021,Z 983.629,A -85,B 0,C 180,E1 -24513.012,E2 -24513.012} C_VEL
LIN {X 0,Y 265.44,Z 999.826,A -85,B 0,C 180,E1 -24516.644,E2 -24516.644} C_VEL
LIN {X 0,Y 254.149,Z 1012.603,A -85,B 0,C 180,E1 -24520.248,E2 -24520.248} C_VEL
LIN {X 0,Y 241.908,Z 1025.908,A -85,B 0,C 180,E1 -24525.024,E2 -24525.024} C_VEL
LIN {X 0,Y 232.664,Z 1035.795,A -85,B 0,C 180,E1 -24529.539,E2 -24529.539} C_VEL
LIN {X 0,Y 223.13,Z 1046.149,A -85,B 0,C 180,E1 -24535.623,E2 -24535.623} C_VEL
LIN {X 0,Y 216.861,Z 1053.354,A -85,B 0,C 180,E1 -24541.169,E2 -24541.169} C_VEL
LIN {X 0,Y 211.85,Z 1059.921,A -85,B 0,C 180,E1 -24547.816,E2 -24547.816} C_VEL
LIN {X 0,Y 209.24,Z 1064.203,A -85,B 0,C 180,E1 -24553.909,E2 -24553.909} C_VEL
LIN {X 0,Y 208.181,Z 1066.945,A -85,B 0,C 180,E1 -24559.484,E2 -24559.484} C_VEL
LIN {X 0,Y 207.983,Z 1068.651,A -85,B 0,C 180,E1 -24565.312,E2 -24565.312} C_VEL
LIN {X 0,Y 208.025,Z 1069.02,A -85,B 0,C 180,E1 -24570.551,E2 -24570.551} C_VEL
LIN {X 0,Y 207.986,Z 1068.358,A -85,B 0,C 180,E1 -24575.794,E2 -24575.794} C_VEL
LIN {X 0,Y 208.24,Z 1066.685,A -85,B 0,C 180,E1 -24581.073,E2 -24581.073} C_VEL
LIN {X 0,Y 209.41,Z 1063.84,A -85,B 0,C 180,E1 -24586.648,E2 -24586.648} C_VEL
LIN {X 0,Y 212.505,Z 1058.955,A -85,B 0,C 180,E1 -24593.281,E2 -24593.281} C_VEL
LIN {X 0,Y 217.472,Z 1052.541,A -85,B 0,C 180,E1 -24599.469,E2 -24599.469} C_VEL
LIN {X 0,Y 224.583,Z 1044.541,A -85,B 0,C 180,E1 -24605.437,E2 -24605.437} C_VEL
LIN {X 0,Y 233.517,Z 1034.764,A -85,B 0,C 180,E1 -24610.929,E2 -24610.929} C_VEL
LIN {X 0,Y 243.911,Z 1023.708,A -85,B 0,C 180,E1 -24615.84,E2 -24615.84} C_VEL
LIN {X 0,Y 255.273,Z 1011.175,A -85,B 0,C 180,E1 -24620.149,E2 -24620.149} C_VEL
LIN {X 0,Y 266.673,Z 998.245,A -85,B 0,C 180,E1 -24623.72,E2 -24623.72} C_VEL
LIN {X 0,Y 279.676,Z 982.573,A -85,B 0,C 180,E1 -24627.157,E2 -24627.157} C_VEL
LIN {X 0,Y 290.739,Z 968.335,A -85,B 0,C 180,E1 -24629.68,E2 -24629.68} C_VEL
LIN {X 0,Y 303.822,Z 950.252,A -85,B 0,C 180,E1 -24632.287,E2 -24632.287} C_VEL
LIN {X 0,Y 315.546,Z 932.311,A -85,B 0,C 180,E1 -24634.357,E2 -24634.357} C_VEL
LIN {X 0,Y 327.418,Z 912.47,A -85,B 0,C 180,E1 -24636.227,E2 -24636.227} C_VEL
LIN {X 0,Y 338.165,Z 892.055,A -85,B 0,C 180,E1 -24637.761,E2 -24637.761} C_VEL
LIN {X 0,Y 347.974,Z 871.231,A -85,B 0,C 180,E1 -24639.047,E2 -24639.047} C_VEL
LIN {X 0,Y 357.165,Z 848.407,A -85,B 0,C 180,E1 -24640.158,E2 -24640.158} C_VEL
LIN {X 0,Y 364.814,Z 826.369,A -85,B 0,C 180,E1 -24641.011,E2 -24641.011} C_VEL
LIN {X 0,Y 371.652,Z 802.115,A -85,B 0,C 180,E1 -24641.732,E2 -24641.732} C_VEL
LIN {X 0,Y 376.535,Z 780.405,A -85,B 0,C 180,E1 -24642.236,E2 -24642.236} C_VEL
LIN {X 0,Y 380.746,Z 754.035,A -85,B 0,C 180,E1 -24642.725,E2 -24642.725} C_VEL
LIN {X 0,Y 396.863,Z 591.973,A -85,B 0,C 180,E1 -24645.183,E2 -24645.183} C_VEL
LIN {X 0,Y 394.714,Z 587.291,A -85,B 0,C 180,E1 -24646.747,E2 -24646.747} C_VEL
LIN {X 0,Y 391.346,Z 580.637,A -85,B 0,C 180,E1 -24649.623,E2 -24649.623} C_VEL
LIN {X 0,Y 389.395,Z 576.922,A -85,B 0,C 180,E1 -24651.732,E2 -24651.732} C_VEL
LIN {X 0,Y 387.595,Z 573.29,A -85,B 0,C 180,E1 -24654.374,E2 -24654.374} C_VEL
LIN {X 0,Y 386.11,Z 569.031,A -85,B 0,C 180,E1 -24660.297,E2 -24660.297} C_VEL
LIN {X 0,Y 387.907,Z 573.936,A -85,B 0,C 180,E1 -24666.587,E2 -24666.587} C_VEL
LIN {X 0,Y 390.17,Z 578.433,A -85,B 0,C 180,E1 -24669.589,E2 -24669.589} C_VEL
LIN {X 0,Y 392.627,Z 583.166,A -85,B 0,C 180,E1 -24671.979,E2 -24671.979} C_VEL
LIN {X 0,Y 396.416,Z 590.741,A -85,B 0,C 180,E1 -24674.909,E2 -24674.909} C_VEL
LIN {X 0,Y 396.815,Z 591.739,A -85,B 0,C 180,E1 -24675.195,E2 -24675.195} C_VEL
LIN {X 0,Y 381.068,Z 749.259,A -85,B 0,C 180,E1 -24677.57,E2 -24677.57} C_VEL
LIN {X 0,Y 376.791,Z 775.495,A -85,B 0,C 180,E1 -24678.081,E2 -24678.081} C_VEL
LIN {X 0,Y 372.087,Z 796.576,A -85,B 0,C 180,E1 -24678.617,E2 -24678.617} C_VEL
LIN {X 0,Y 365.245,Z 821.003,A -85,B 0,C 180,E1 -24679.422,E2 -24679.422} C_VEL
LIN {X 0,Y 358.184,Z 841.639,A -85,B 0,C 180,E1 -24680.288,E2 -24680.288} C_VEL
LIN {X 0,Y 349.587,Z 863.409,A -85,B 0,C 180,E1 -24681.41,E2 -24681.41} C_VEL
LIN {X 0,Y 339.88,Z 884.23,A -85,B 0,C 180,E1 -24682.738,E2 -24682.738} C_VEL
LIN {X 0,Y 329.976,Z 903.23,A -85,B 0,C 180,E1 -24684.205,E2 -24684.205} C_VEL
LIN {X 0,Y 318.005,Z 923.578,A -85,B 0,C 180,E1 -24686.145,E2 -24686.145} C_VEL
LIN {X 0,Y 307.133,Z 940.278,A -85,B 0,C 180,E1 -24688.085,E2 -24688.085} C_VEL
LIN {X 0,Y 293.449,Z 959.37,A -85,B 0,C 180,E1 -24690.834,E2 -24690.834} C_VEL
LIN {X 0,Y 282.463,Z 973.435,A -85,B 0,C 180,E1 -24693.341,E2 -24693.341} C_VEL
LIN {X 0,Y 269.526,Z 988.942,A -85,B 0,C 180,E1 -24696.744,E2 -24696.744} C_VEL
LIN {X 0,Y 257.82,Z 1001.978,A -85,B 0,C 180,E1 -24700.366,E2 -24700.366} C_VEL
LIN {X 0,Y 246.186,Z 1014.482,A -85,B 0,C 180,E1 -24704.703,E2 -24704.703} C_VEL
LIN {X 0,Y 235.717,Z 1025.205,A -85,B 0,C 180,E1 -24709.533,E2 -24709.533} C_VEL
LIN {X 0,Y 226.523,Z 1034.738,A -85,B 0,C 180,E1 -24714.983,E2 -24714.983} C_VEL
LIN {X 0,Y 219.219,Z 1042.336,A -85,B 0,C 180,E1 -24720.788,E2 -24720.788} C_VEL
LIN {X 0,Y 213.892,Z 1048.456,A -85,B 0,C 180,E1 -24726.879,E2 -24726.879} C_VEL
LIN {X 0,Y 210.338,Z 1053.079,A -85,B 0,C 180,E1 -24733.428,E2 -24733.428} C_VEL
LIN {X 0,Y 208.734,Z 1055.807,A -85,B 0,C 180,E1 -24739.115,E2 -24739.115} C_VEL
LIN {X 0,Y 208.122,Z 1057.494,A -85,B 0,C 180,E1 -24745.039,E2 -24745.039} C_VEL
LIN {X 0,Y 208.032,Z 1057.901,A -85,B 0,C 180,E1 -24750.826,E2 -24750.826} C_VEL
LIN {X 0,Y 208.178,Z 1057.246,A -85,B 0,C 180,E1 -24756.153,E2 -24756.153} C_VEL
LIN {X 0,Y 208.861,Z 1055.584,A -85,B 0,C 180,E1 -24761.6,E2 -24761.6} C_VEL
LIN {X 0,Y 210.764,Z 1052.544,A -85,B 0,C 180,E1 -24767.676,E2 -24767.676} C_VEL
LIN {X 0,Y 214.617,Z 1047.594,A -85,B 0,C 180,E1 -24774.204,E2 -24774.204} C_VEL
LIN {X 0,Y 219.7,Z 1041.9,A -85,B 0,C 180,E1 -24779.741,E2 -24779.741} C_VEL
LIN {X 0,Y 227.512,Z 1033.763,A -85,B 0,C 180,E1 -24785.769,E2 -24785.769} C_VEL
LIN {X 0,Y 236.046,Z 1024.982,A -85,B 0,C 180,E1 -24790.719,E2 -24790.719} C_VEL
LIN {X 0,Y 246.573,Z 1014.22,A -85,B 0,C 180,E1 -24795.537,E2 -24795.537} C_VEL
LIN {X 0,Y 257.996,Z 1001.951,A -85,B 0,C 180,E1 -24799.774,E2 -24799.774} C_VEL
LIN {X 0,Y 270.014,Z 988.593,A -85,B 0,C 180,E1 -24803.473,E2 -24803.473} C_VEL
LIN {X 0,Y 282.338,Z 973.827,A -85,B 0,C 180,E1 -24806.706,E2 -24806.706} C_VEL
LIN {X 0,Y 293.634,Z 959.387,A -85,B 0,C 180,E1 -24809.284,E2 -24809.284} C_VEL
LIN {X 0,Y 307.397,Z 940.201,A -85,B 0,C 180,E1 -24812.042,E2 -24812.042} C_VEL
LIN {X 0,Y 318.244,Z 923.554,A -85,B 0,C 180,E1 -24813.973,E2 -24813.973} C_VEL
LIN {X 0,Y 330.228,Z 903.198,A -85,B 0,C 180,E1 -24815.91,E2 -24815.91} C_VEL
LIN {X 0,Y 339.801,Z 884.872,A -85,B 0,C 180,E1 -24817.326,E2 -24817.326} C_VEL
LIN {X 0,Y 349.45,Z 864.256,A -85,B 0,C 180,E1 -24818.648,E2 -24818.648} C_VEL
LIN {X 0,Y 358.345,Z 841.877,A -85,B 0,C 180,E1 -24819.806,E2 -24819.806} C_VEL
LIN {X 0,Y 365.534,Z 820.898,A -85,B 0,C 180,E1 -24820.686,E2 -24820.686} C_VEL
LIN {X 0,Y 372.434,Z 796.204,A -85,B 0,C 180,E1 -24821.497,E2 -24821.497} C_VEL
LIN {X 0,Y 377.163,Z 774.936,A -85,B 0,C 180,E1 -24822.035,E2 -24822.035} C_VEL
LIN {X 0,Y 381.454,Z 748.203,A -85,B 0,C 180,E1 -24822.55,E2 -24822.55} C_VEL
LIN {X 0,Y 397.072,Z 591.697,A -85,B 0,C 180,E1 -24824.917,E2 -24824.917} C_VEL
LIN {X 0,Y 393.162,Z 583.892,A -85,B 0,C 180,E1 -24827.888,E2 -24827.888} C_VEL
LIN {X 0,Y 390.926,Z 579.693,A -85,B 0,C 180,E1 -24829.984,E2 -24829.984} C_VEL
LIN {X 0,Y 389.526,Z 576.964,A -85,B 0,C 180,E1 -24831.586,E2 -24831.586} C_VEL
LIN {X 0,Y 387.791,Z 573.386,A -85,B 0,C 180,E1 -24834.229,E2 -24834.229} C_VEL
LIN {X 0,Y 386.376,Z 569.819,A -85,B 0,C 180,E1 -24840,E2 -24840} C_VEL
LIN {X 0,Y 387.889,Z 573.488,A -85,B 0,C 180,E1 -24845.604,E2 -24845.604} C_VEL
LIN {X 0,Y 388.403,Z 575.002,A -85,B 0,C 180,E1 -24846.551,E2 -24846.551} C_VEL
LIN {X 0,Y 388.923,Z 579.017,A -85,B 0,C 180,E1 -24847.721,E2 -24847.721} C_VEL
LIN {X 0,Y 390.018,Z 587.241,A -85,B 0,C 180,E1 -24849.713,E2 -24849.713} C_VEL
LIN {X 0,Y 390.552,Z 588.948,A -85,B 0,C 180,E1 -24850.323,E2 -24850.323} C_VEL
LIN {X 0,Y 394.102,Z 596.247,A -85,B 0,C 180,E1 -24853.386,E2 -24853.386} C_VEL
LIN {X 0,Y 394.581,Z 597.586,A -85,B 0,C 180,E1 -24853.771,E2 -24853.771} C_VEL
LIN {X 0,Y 378.539,Z 755.173,A -85,B 0,C 180,E1 -24856.123,E2 -24856.123} C_VEL
LIN {X 0,Y 374.103,Z 781.719,A -85,B 0,C 180,E1 -24856.612,E2 -24856.612} C_VEL
LIN {X 0,Y 369.102,Z 803.358,A -85,B 0,C 180,E1 -24857.106,E2 -24857.106} C_VEL
LIN {X 0,Y 361.86,Z 828.136,A -85,B 0,C 180,E1 -24857.839,E2 -24857.839} C_VEL
LIN {X 0,Y 354.527,Z 848.792,A -85,B 0,C 180,E1 -24858.623,E2 -24858.623} C_VEL
LIN {X 0,Y 344.94,Z 872.005,A -85,B 0,C 180,E1 -24859.735,E2 -24859.735} C_VEL
LIN {X 0,Y 335.16,Z 892.342,A -85,B 0,C 180,E1 -24860.968,E2 -24860.968} C_VEL
LIN {X 0,Y 323.984,Z 913.071,A -85,B 0,C 180,E1 -24862.501,E2 -24862.501} C_VEL
LIN {X 0,Y 312.121,Z 932.4,A -85,B 0,C 180,E1 -24864.297,E2 -24864.297} C_VEL
LIN {X 0,Y 300.119,Z 950.311,A -85,B 0,C 180,E1 -24866.335,E2 -24866.335} C_VEL
LIN {X 0,Y 287.425,Z 967.409,A -85,B 0,C 180,E1 -24868.758,E2 -24868.758} C_VEL
LIN {X 0,Y 276.006,Z 981.706,A -85,B 0,C 180,E1 -24871.244,E2 -24871.244} C_VEL
LIN {X 0,Y 262.534,Z 997.482,A -85,B 0,C 180,E1 -24874.648,E2 -24874.648} C_VEL
LIN {X 0,Y 250.659,Z 1010.456,A -85,B 0,C 180,E1 -24878.201,E2 -24878.201} C_VEL
LIN {X 0,Y 238.75,Z 1023.065,A -85,B 0,C 180,E1 -24882.516,E2 -24882.516} C_VEL
LIN {X 0,Y 227.577,Z 1034.384,A -85,B 0,C 180,E1 -24887.573,E2 -24887.573} C_VEL
LIN {X 0,Y 218.173,Z 1044.101,A -85,B 0,C 180,E1 -24893.103,E2 -24893.103} C_VEL
LIN {X 0,Y 210.399,Z 1052.289,A -85,B 0,C 180,E1 -24899.337,E2 -24899.337} C_VEL
LIN {X 0,Y 205.156,Z 1058.527,A -85,B 0,C 180,E1 -24905.526,E2 -24905.526} C_VEL
LIN {X 0,Y 201.694,Z 1063.49,A -85,B 0,C 180,E1 -24912.398,E2 -24912.398} C_VEL
LIN {X 0,Y 200.326,Z 1066.375,A -85,B 0,C 180,E1 -24918.191,E2 -24918.191} C_VEL
LIN {X 0,Y 199.986,Z 1068.086,A -85,B 0,C 180,E1 -24923.685,E2 -24923.685} C_VEL
LIN {X 0,Y 200.023,Z 1068.765,A -85,B 0,C 180,E1 -24928.854,E2 -24928.854} C_VEL
LIN {X 0,Y 199.989,Z 1068.52,A -85,B 0,C 180,E1 -24934.014,E2 -24934.014} C_VEL
LIN {X 0,Y 200.136,Z 1067.058,A -85,B 0,C 180,E1 -24940.07,E2 -24940.07} C_VEL
LIN {X 0,Y 201.318,Z 1064.117,A -85,B 0,C 180,E1 -24946.445,E2 -24946.445} C_VEL
LIN {X 0,Y 203.921,Z 1060.085,A -85,B 0,C 180,E1 -24952.486,E2 -24952.486} C_VEL
LIN {X 0,Y 209.497,Z 1053.25,A -85,B 0,C 180,E1 -24959.76,E2 -24959.76} C_VEL
LIN {X 0,Y 215.984,Z 1046.21,A -85,B 0,C 180,E1 -24965.358,E2 -24965.358} C_VEL
LIN {X 0,Y 225.996,Z 1035.903,A -85,B 0,C 180,E1 -24971.606,E2 -24971.606} C_VEL
LIN {X 0,Y 235.813,Z 1025.866,A -85,B 0,C 180,E1 -24976.279,E2 -24976.279} C_VEL
LIN {X 0,Y 248.694,Z 1012.42,A -85,B 0,C 180,E1 -24981.155,E2 -24981.155} C_VEL
LIN {X 0,Y 259.931,Z 1000.148,A -85,B 0,C 180,E1 -24984.638,E2 -24984.638} C_VEL
LIN {X 0,Y 273.219,Z 984.911,A -85,B 0,C 180,E1 -24988.107,E2 -24988.107} C_VEL
LIN {X 0,Y 285.947,Z 969.046,A -85,B 0,C 180,E1 -24990.949,E2 -24990.949} C_VEL
LIN {X 0,Y 298.958,Z 951.688,A -85,B 0,C 180,E1 -24993.466,E2 -24993.466} C_VEL
LIN {X 0,Y 311.308,Z 933.314,A -85,B 0,C 180,E1 -24995.584,E2 -24995.584} C_VEL
LIN {X 0,Y 322.554,Z 915.042,A -85,B 0,C 180,E1 -24997.308,E2 -24997.308} C_VEL
LIN {X 0,Y 334.31,Z 893.536,A -85,B 0,C 180,E1 -24998.933,E2 -24998.933} C_VEL
LIN {X 0,Y 343.472,Z 874.624,A -85,B 0,C 180,E1 -25000.1,E2 -25000.1} C_VEL
LIN {X 0,Y 353.652,Z 850.453,A -85,B 0,C 180,E1 -25001.29,E2 -25001.29} C_VEL
LIN {X 0,Y 361.017,Z 829.883,A -85,B 0,C 180,E1 -25002.084,E2 -25002.084} C_VEL
LIN {X 0,Y 368.253,Z 805.713,A -85,B 0,C 180,E1 -25002.82,E2 -25002.82} C_VEL
LIN {X 0,Y 373.482,Z 783.429,A -85,B 0,C 180,E1 -25003.34,E2 -25003.34} C_VEL
LIN {X 0,Y 377.853,Z 758.646,A -85,B 0,C 180,E1 -25003.808,E2 -25003.808} C_VEL
LIN {X 0,Y 383.618,Z 703.877,A -85,B 0,C 180,E1 -25004.647,E2 -25004.647} C_VEL
LIN {X 0,Y 394.322,Z 597.081,A -85,B 0,C 180,E1 -25006.244,E2 -25006.244} C_VEL
LIN {X 0,Y 391.102,Z 590.543,A -85,B 0,C 180,E1 -25008.871,E2 -25008.871} C_VEL
LIN {X 0,Y 388.54,Z 585.184,A -85,B 0,C 180,E1 -25011.565,E2 -25011.565} C_VEL
LIN {X 0,Y 386.531,Z 581.173,A -85,B 0,C 180,E1 -25014.508,E2 -25014.508} C_VEL
LIN {X 0,Y 385.129,Z 577.015,A -85,B 0,C 180,E1 -25020.298,E2 -25020.298} C_VEL
LIN {X 0,Y 386.79,Z 581.745,A -85,B 0,C 180,E1 -25026.382,E2 -25026.382} C_VEL
LIN {X 0,Y 388.979,Z 586.268,A -85,B 0,C 180,E1 -25029.394,E2 -25029.394} C_VEL
LIN {X 0,Y 391.379,Z 591.028,A -85,B 0,C 180,E1 -25031.793,E2 -25031.793} C_VEL
LIN {X 0,Y 394.277,Z 597.06,A -85,B 0,C 180,E1 -25034.149,E2 -25034.149} C_VEL
LIN {X 0,Y 378.729,Z 749.495,A -85,B 0,C 180,E1 -25036.416,E2 -25036.416} C_VEL
LIN {X 0,Y 374.384,Z 775.722,A -85,B 0,C 180,E1 -25036.916,E2 -25036.916} C_VEL
LIN {X 0,Y 369.605,Z 796.802,A -85,B 0,C 180,E1 -25037.439,E2 -25037.439} C_VEL
LIN {X 0,Y 362.655,Z 821.225,A -85,B 0,C 180,E1 -25038.226,E2 -25038.226} C_VEL
LIN {X 0,Y 355.477,Z 841.861,A -85,B 0,C 180,E1 -25039.073,E2 -25039.073} C_VEL
LIN {X 0,Y 346.586,Z 863.948,A -85,B 0,C 180,E1 -25040.188,E2 -25040.188} C_VEL
LIN {X 0,Y 336.841,Z 884.451,A -85,B 0,C 180,E1 -25041.472,E2 -25041.472} C_VEL
LIN {X 0,Y 327.251,Z 902.513,A -85,B 0,C 180,E1 -25042.833,E2 -25042.833} C_VEL
LIN {X 0,Y 314.901,Z 923.195,A -85,B 0,C 180,E1 -25044.753,E2 -25044.753} C_VEL
LIN {X 0,Y 303.764,Z 939.948,A -85,B 0,C 180,E1 -25046.66,E2 -25046.66} C_VEL
LIN {X 0,Y 289.97,Z 958.803,A -85,B 0,C 180,E1 -25049.318,E2 -25049.318} C_VEL
LIN {X 0,Y 278.05,Z 973.656,A -85,B 0,C 180,E1 -25051.933,E2 -25051.933} C_VEL
LIN {X 0,Y 264.705,Z 989.163,A -85,B 0,C 180,E1 -25055.323,E2 -25055.323} C_VEL
LIN {X 0,Y 252.903,Z 1001.861,A -85,B 0,C 180,E1 -25058.843,E2 -25058.843} C_VEL
LIN {X 0,Y 241.009,Z 1014.169,A -85,B 0,C 180,E1 -25063.099,E2 -25063.099} C_VEL
LIN {X 0,Y 229.738,Z 1025.219,A -85,B 0,C 180,E1 -25068.095,E2 -25068.095} C_VEL
LIN {X 0,Y 220.222,Z 1034.572,A -85,B 0,C 180,E1 -25073.503,E2 -25073.503} C_VEL
LIN {X 0,Y 212.286,Z 1042.367,A -85,B 0,C 180,E1 -25079.537,E2 -25079.537} C_VEL
LIN {X 0,Y 206.814,Z 1048.179,A -85,B 0,C 180,E1 -25085.431,E2 -25085.431} C_VEL
LIN {X 0,Y 202.684,Z 1053.142,A -85,B 0,C 180,E1 -25092.487,E2 -25092.487} C_VEL
LIN {X 0,Y 200.906,Z 1055.85,A -85,B 0,C 180,E1 -25098.226,E2 -25098.226} C_VEL
LIN {X 0,Y 200.175,Z 1057.511,A -85,B 0,C 180,E1 -25103.979,E2 -25103.979} C_VEL
LIN {X 0,Y 200.038,Z 1058.168,A -85,B 0,C 180,E1 -25110,E2 -25110} C_VEL
LIN {X 0,Y 200.173,Z 1057.546,A -85,B 0,C 180,E1 -25116.022,E2 -25116.022} C_VEL
LIN {X 0,Y 200.891,Z 1055.909,A -85,B 0,C 180,E1 -25121.775,E2 -25121.775} C_VEL
LIN {X 0,Y 202.775,Z 1053.07,A -85,B 0,C 180,E1 -25127.802,E2 -25127.802} C_VEL
LIN {X 0,Y 207.185,Z 1047.812,A -85,B 0,C 180,E1 -25135.132,E2 -25135.132} C_VEL
LIN {X 0,Y 212.615,Z 1042.118,A -85,B 0,C 180,E1 -25140.838,E2 -25140.838} C_VEL
LIN {X 0,Y 220.894,Z 1033.981,A -85,B 0,C 180,E1 -25147.016,E2 -25147.016} C_VEL
LIN {X 0,Y 229.875,Z 1025.2,A -85,B 0,C 180,E1 -25152.056,E2 -25152.056} C_VEL
LIN {X 0,Y 240.885,Z 1014.438,A -85,B 0,C 180,E1 -25156.934,E2 -25156.934} C_VEL
LIN {X 0,Y 252.771,Z 1002.168,A -85,B 0,C 180,E1 -25161.195,E2 -25161.195} C_VEL
LIN {X 0,Y 265.216,Z 988.81,A -85,B 0,C 180,E1 -25164.896,E2 -25164.896} C_VEL
LIN {X 0,Y 277.914,Z 974.062,A -85,B 0,C 180,E1 -25168.113,E2 -25168.113} C_VEL
LIN {X 0,Y 289.211,Z 960.03,A -85,B 0,C 180,E1 -25170.603,E2 -25170.603} C_VEL
LIN {X 0,Y 302.875,Z 941.571,A -85,B 0,C 180,E1 -25173.254,E2 -25173.254} C_VEL
LIN {X 0,Y 313.987,Z 924.976,A -85,B 0,C 180,E1 -25175.174,E2 -25175.174} C_VEL
LIN {X 0,Y 325.814,Z 905.6,A -85,B 0,C 180,E1 -25177.024,E2 -25177.024} C_VEL
LIN {X 0,Y 336.301,Z 886.009,A -85,B 0,C 180,E1 -25178.53,E2 -25178.53} C_VEL
LIN {X 0,Y 345.763,Z 866.258,A -85,B 0,C 180,E1 -25179.785,E2 -25179.785} C_VEL
LIN {X 0,Y 355.065,Z 843.648,A -85,B 0,C 180,E1 -25180.952,E2 -25180.952} C_VEL
LIN {X 0,Y 362.37,Z 822.872,A -85,B 0,C 180,E1 -25181.815,E2 -25181.815} C_VEL
LIN {X 0,Y 369.808,Z 797.056,A -85,B 0,C 180,E1 -25182.656,E2 -25182.656} C_VEL
LIN {X 0,Y 374.609,Z 775.917,A -85,B 0,C 180,E1 -25183.182,E2 -25183.182} C_VEL
LIN {X 0,Y 378.962,Z 749.785,A -85,B 0,C 180,E1 -25183.681,E2 -25183.681} C_VEL
LIN {X 0,Y 391.906,Z 623.162,A -85,B 0,C 180,E1 -25185.571,E2 -25185.571} C_VEL
LIN {X 0,Y 394.526,Z 597.237,A -85,B 0,C 180,E1 -25185.956,E2 -25185.956} C_VEL
LIN {X 0,Y 391.344,Z 590.649,A -85,B 0,C 180,E1 -25188.579,E2 -25188.579} C_VEL
LIN {X 0,Y 388.546,Z 585.036,A -85,B 0,C 180,E1 -25191.565,E2 -25191.565} C_VEL
LIN {X 0,Y 386.732,Z 581.269,A -85,B 0,C 180,E1 -25194.362,E2 -25194.362} C_VEL
LIN {X 0,Y 385.398,Z 577.786,A -85,B 0,C 180,E1 -25200,E2 -25200} C_VEL
LIN {X 0,Y 387.031,Z 581.872,A -85,B 0,C 180,E1 -25205.857,E2 -25205.857} C_VEL
LIN {X 0,Y 389.179,Z 586.289,A -85,B 0,C 180,E1 -25208.868,E2 -25208.868} C_VEL
LIN {X 0,Y 390.552,Z 588.948,A -85,B 0,C 180,E1 -25210.323,E2 -25210.323} C_VEL
LIN {X 0,Y 391.415,Z 592.058,A -85,B 0,C 180,E1 -25211.271,E2 -25211.271} C_VEL
LIN {X 0,Y 391.987,Z 596.651,A -85,B 0,C 180,E1 -25212.072,E2 -25212.072} C_VEL
LIN {X 0,Y 392.108,Z 601.785,A -85,B 0,C 180,E1 -25212.578,E2 -25212.578} C_VEL
LIN {X 0,Y 391.837,Z 606.197,A -85,B 0,C 180,E1 -25212.76,E2 -25212.76} C_VEL
LIN {X 0,Y 376.388,Z 754.98,A -85,B 0,C 180,E1 -25214.949,E2 -25214.949} C_VEL
LIN {X 0,Y 371.889,Z 781.504,A -85,B 0,C 180,E1 -25215.426,E2 -25215.426} C_VEL
LIN {X 0,Y 366.815,Z 803.163,A -85,B 0,C 180,E1 -25215.905,E2 -25215.905} C_VEL
LIN {X 0,Y 359.473,Z 827.928,A -85,B 0,C 180,E1 -25216.616,E2 -25216.616} C_VEL
LIN {X 0,Y 352.031,Z 848.584,A -85,B 0,C 180,E1 -25217.377,E2 -25217.377} C_VEL
LIN {X 0,Y 342.537,Z 871.277,A -85,B 0,C 180,E1 -25218.432,E2 -25218.432} C_VEL
LIN {X 0,Y 332.764,Z 891.315,A -85,B 0,C 180,E1 -25219.609,E2 -25219.609} C_VEL
LIN {X 0,Y 322.045,Z 910.954,A -85,B 0,C 180,E1 -25221.009,E2 -25221.009} C_VEL
LIN {X 0,Y 309.564,Z 931.096,A -85,B 0,C 180,E1 -25222.805,E2 -25222.805} C_VEL
LIN {X 0,Y 298.13,Z 947.86,A -85,B 0,C 180,E1 -25224.646,E2 -25224.646} C_VEL
LIN {X 0,Y 283.755,Z 966.952,A -85,B 0,C 180,E1 -25227.264,E2 -25227.264} C_VEL
LIN {X 0,Y 271.654,Z 981.685,A -85,B 0,C 180,E1 -25229.795,E2 -25229.795} C_VEL
LIN {X 0,Y 257.253,Z 997.972,A -85,B 0,C 180,E1 -25233.315,E2 -25233.315} C_VEL
LIN {X 0,Y 245.004,Z 1010.879,A -85,B 0,C 180,E1 -25236.879,E2 -25236.879} C_VEL
LIN {X 0,Y 232.112,Z 1023.901,A -85,B 0,C 180,E1 -25241.448,E2 -25241.448} C_VEL
LIN {X 0,Y 221.258,Z 1034.422,A -85,B 0,C 180,E1 -25246.257,E2 -25246.257} C_VEL
LIN {X 0,Y 211.204,Z 1044.267,A -85,B 0,C 180,E1 -25252.015,E2 -25252.015} C_VEL
LIN {X 0,Y 203.234,Z 1052.166,A -85,B 0,C 180,E1 -25258.235,E2 -25258.235} C_VEL
LIN {X 0,Y 197.485,Z 1058.569,A -85,B 0,C 180,E1 -25264.83,E2 -25264.83} C_VEL
LIN {X 0,Y 193.805,Z 1063.437,A -85,B 0,C 180,E1 -25271.967,E2 -25271.967} C_VEL
LIN {X 0,Y 192.346,Z 1066.276,A -85,B 0,C 180,E1 -25277.998,E2 -25277.998} C_VEL
LIN {X 0,Y 191.988,Z 1068.038,A -85,B 0,C 180,E1 -25284.126,E2 -25284.126} C_VEL
LIN {X 0,Y 192.032,Z 1068.62,A -85,B 0,C 180,E1 -25289.701,E2 -25289.701} C_VEL
LIN {X 0,Y 191.988,Z 1068.14,A -85,B 0,C 180,E1 -25295.379,E2 -25295.379} C_VEL
LIN {X 0,Y 192.307,Z 1066.37,A -85,B 0,C 180,E1 -25301.699,E2 -25301.699} C_VEL
LIN {X 0,Y 193.698,Z 1063.568,A -85,B 0,C 180,E1 -25307.732,E2 -25307.732} C_VEL
LIN {X 0,Y 197.283,Z 1058.775,A -85,B 0,C 180,E1 -25314.876,E2 -25314.876} C_VEL
LIN {X 0,Y 203.016,Z 1052.321,A -85,B 0,C 180,E1 -25321.564,E2 -25321.564} C_VEL
LIN {X 0,Y 210.808,Z 1044.545,A -85,B 0,C 180,E1 -25327.724,E2 -25327.724} C_VEL
LIN {X 0,Y 220.769,Z 1034.785,A -85,B 0,C 180,E1 -25333.505,E2 -25333.505} C_VEL
LIN {X 0,Y 231.439,Z 1024.412,A -85,B 0,C 180,E1 -25338.292,E2 -25338.292} C_VEL
LIN {X 0,Y 244.371,Z 1011.372,A -85,B 0,C 180,E1 -25342.928,E2 -25342.928} C_VEL
LIN {X 0,Y 255.899,Z 999.217,A -85,B 0,C 180,E1 -25346.332,E2 -25346.332} C_VEL
LIN {X 0,Y 270.373,Z 982.981,A -85,B 0,C 180,E1 -25349.925,E2 -25349.925} C_VEL
LIN {X 0,Y 282.793,Z 967.89,A -85,B 0,C 180,E1 -25352.557,E2 -25352.557} C_VEL
LIN {X 0,Y 296.553,Z 949.807,A -85,B 0,C 180,E1 -25355.092,E2 -25355.092} C_VEL
LIN {X 0,Y 308.42,Z 932.48,A -85,B 0,C 180,E1 -25357.031,E2 -25357.031} C_VEL
LIN {X 0,Y 320.37,Z 913.409,A -85,B 0,C 180,E1 -25358.774,E2 -25358.774} C_VEL
LIN {X 0,Y 331.857,Z 892.581,A -85,B 0,C 180,E1 -25360.29,E2 -25360.29} C_VEL
LIN {X 0,Y 341.657,Z 872.595,A -85,B 0,C 180,E1 -25361.48,E2 -25361.48} C_VEL
LIN {X 0,Y 351.576,Z 849.096,A -85,B 0,C 180,E1 -25362.586,E2 -25362.586} C_VEL
LIN {X 0,Y 359.013,Z 828.5,A -85,B 0,C 180,E1 -25363.35,E2 -25363.35} C_VEL
LIN {X 0,Y 366.571,Z 803.071,A -85,B 0,C 180,E1 -25364.083,E2 -25364.083} C_VEL
LIN {X 0,Y 371.621,Z 781.492,A -85,B 0,C 180,E1 -25364.562,E2 -25364.562} C_VEL
LIN {X 0,Y 376.113,Z 754.977,A -85,B 0,C 180,E1 -25365.04,E2 -25365.04} C_VEL
LIN {X 0,Y 391.908,Z 602.645,A -85,B 0,C 180,E1 -25367.287,E2 -25367.287} C_VEL
LIN {X 0,Y 388.699,Z 595.885,A -85,B 0,C 180,E1 -25370.225,E2 -25370.225} C_VEL
LIN {X 0,Y 386.951,Z 592.329,A -85,B 0,C 180,E1 -25372.278,E2 -25372.278} C_VEL
LIN {X 0,Y 385.385,Z 588.965,A -85,B 0,C 180,E1 -25374.79,E2 -25374.79} C_VEL
LIN {X 0,Y 384.146,Z 585.023,A -85,B 0,C 180,E1 -25380.298,E2 -25380.298} C_VEL
LIN {X 0,Y 385.716,Z 589.67,A -85,B 0,C 180,E1 -25386.251,E2 -25386.251} C_VEL
LIN {X 0,Y 387.733,Z 593.959,A -85,B 0,C 180,E1 -25389.126,E2 -25389.126} C_VEL
LIN {X 0,Y 390.056,Z 598.73,A -85,B 0,C 180,E1 -25391.534,E2 -25391.534} C_VEL
LIN {X 0,Y 391.832,Z 602.757,A -85,B 0,C 180,E1 -25393.094,E2 -25393.094} C_VEL
LIN {X 0,Y 376.548,Z 749.714,A -85,B 0,C 180,E1 -25395.248,E2 -25395.248} C_VEL
LIN {X 0,Y 372.133,Z 775.949,A -85,B 0,C 180,E1 -25395.737,E2 -25395.737} C_VEL
LIN {X 0,Y 367.255,Z 797.134,A -85,B 0,C 180,E1 -25396.249,E2 -25396.249} C_VEL
LIN {X 0,Y 359.793,Z 822.728,A -85,B 0,C 180,E1 -25397.06,E2 -25397.06} C_VEL
LIN {X 0,Y 352.504,Z 843.209,A -85,B 0,C 180,E1 -25397.889,E2 -25397.889} C_VEL
LIN {X 0,Y 343.185,Z 865.66,A -85,B 0,C 180,E1 -25399.013,E2 -25399.013} C_VEL
LIN {X 0,Y 333.555,Z 885.478,A -85,B 0,C 180,E1 -25400.237,E2 -25400.237} C_VEL
LIN {X 0,Y 322.863,Z 905.132,A -85,B 0,C 180,E1 -25401.708,E2 -25401.708} C_VEL
LIN {X 0,Y 310.795,Z 924.624,A -85,B 0,C 180,E1 -25403.523,E2 -25403.523} C_VEL
LIN {X 0,Y 299.389,Z 941.331,A -85,B 0,C 180,E1 -25405.415,E2 -25405.415} C_VEL
LIN {X 0,Y 285.426,Z 959.812,A -85,B 0,C 180,E1 -25408.019,E2 -25408.019} C_VEL
LIN {X 0,Y 273.106,Z 974.714,A -85,B 0,C 180,E1 -25410.641,E2 -25410.641} C_VEL
LIN {X 0,Y 258.723,Z 990.77,A -85,B 0,C 180,E1 -25414.204,E2 -25414.204} C_VEL
LIN {X 0,Y 247.221,Z 1002.709,A -85,B 0,C 180,E1 -25417.559,E2 -25417.559} C_VEL
LIN {X 0,Y 234.357,Z 1015.431,A -85,B 0,C 180,E1 -25422.066,E2 -25422.066} C_VEL
LIN {X 0,Y 223.295,Z 1025.804,A -85,B 0,C 180,E1 -25426.878,E2 -25426.878} C_VEL
LIN {X 0,Y 213.271,Z 1035.179,A -85,B 0,C 180,E1 -25432.448,E2 -25432.448} C_VEL
LIN {X 0,Y 204.999,Z 1042.832,A -85,B 0,C 180,E1 -25438.602,E2 -25438.602} C_VEL
LIN {X 0,Y 198.963,Z 1048.894,A -85,B 0,C 180,E1 -25445.03,E2 -25445.03} C_VEL
LIN {X 0,Y 194.816,Z 1053.514,A -85,B 0,C 180,E1 -25452.065,E2 -25452.065} C_VEL
LIN {X 0,Y 192.938,Z 1056.176,A -85,B 0,C 180,E1 -25458.036,E2 -25458.036} C_VEL
LIN {X 0,Y 192.175,Z 1057.791,A -85,B 0,C 180,E1 -25464.027,E2 -25464.027} C_VEL
LIN {X 0,Y 192.041,Z 1058.382,A -85,B 0,C 180,E1 -25470,E2 -25470} C_VEL
LIN {X 0,Y 192.191,Z 1057.76,A -85,B 0,C 180,E1 -25476.273,E2 -25476.273} C_VEL
LIN {X 0,Y 192.986,Z 1056.125,A -85,B 0,C 180,E1 -25482.265,E2 -25482.265} C_VEL
LIN {X 0,Y 195.044,Z 1053.286,A -85,B 0,C 180,E1 -25488.533,E2 -25488.533} C_VEL
LIN {X 0,Y 199.809,Z 1048.029,A -85,B 0,C 180,E1 -25496.128,E2 -25496.128} C_VEL
LIN {X 0,Y 205.613,Z 1042.336,A -85,B 0,C 180,E1 -25502.01,E2 -25502.01} C_VEL
LIN {X 0,Y 214.802,Z 1033.801,A -85,B 0,C 180,E1 -25508.592,E2 -25508.592} C_VEL
LIN {X 0,Y 224.325,Z 1024.966,A -85,B 0,C 180,E1 -25513.701,E2 -25513.701} C_VEL
LIN {X 0,Y 236.467,Z 1013.532,A -85,B 0,C 180,E1 -25518.822,E2 -25518.822} C_VEL
LIN {X 0,Y 248.328,Z 1001.758,A -85,B 0,C 180,E1 -25522.868,E2 -25522.868} C_VEL
LIN {X 0,Y 261.339,Z 988.244,A -85,B 0,C 180,E1 -25526.568,E2 -25526.568} C_VEL
LIN {X 0,Y 274.388,Z 973.44,A -85,B 0,C 180,E1 -25529.729,E2 -25529.729} C_VEL
LIN {X 0,Y 286.777,Z 958.41,A -85,B 0,C 180,E1 -25532.327,E2 -25532.327} C_VEL
LIN {X 0,Y 300.457,Z 940.132,A -85,B 0,C 180,E1 -25534.849,E2 -25534.849} C_VEL
LIN {X 0,Y 311.857,Z 923.376,A -85,B 0,C 180,E1 -25536.721,E2 -25536.721} C_VEL
LIN {X 0,Y 324.766,Z 902.16,A -85,B 0,C 180,E1 -25538.644,E2 -25538.644} C_VEL
LIN {X 0,Y 334.264,Z 884.604,A -85,B 0,C 180,E1 -25539.93,E2 -25539.93} C_VEL
LIN {X 0,Y 344.333,Z 863.757,A -85,B 0,C 180,E1 -25541.201,E2 -25541.201} C_VEL
LIN {X 0,Y 353.209,Z 842.048,A -85,B 0,C 180,E1 -25542.267,E2 -25542.267} C_VEL
LIN {X 0,Y 361.106,Z 819.641,A -85,B 0,C 180,E1 -25543.157,E2 -25543.157} C_VEL
LIN {X 0,Y 367.902,Z 795.635,A -85,B 0,C 180,E1 -25543.894,E2 -25543.894} C_VEL
LIN {X 0,Y 372.907,Z 773.555,A -85,B 0,C 180,E1 -25544.418,E2 -25544.418} C_VEL
LIN {X 0,Y 377.042,Z 747.945,A -85,B 0,C 180,E1 -25544.882,E2 -25544.882} C_VEL
LIN {X 0,Y 392.087,Z 602.695,A -85,B 0,C 180,E1 -25547.031,E2 -25547.031} C_VEL
LIN {X 0,Y 389.23,Z 596.603,A -85,B 0,C 180,E1 -25549.641,E2 -25549.641} C_VEL
LIN {X 0,Y 387.211,Z 592.563,A -85,B 0,C 180,E1 -25551.984,E2 -25551.984} C_VEL
LIN {X 0,Y 385.593,Z 589.064,A -85,B 0,C 180,E1 -25554.643,E2 -25554.643} C_VEL
LIN {X 0,Y 384.419,Z 585.76,A -85,B 0,C 180,E1 -25560,E2 -25560} C_VEL
LIN {X 0,Y 385.922,Z 589.677,A -85,B 0,C 180,E1 -25565.65,E2 -25565.65} C_VEL
LIN {X 0,Y 387.996,Z 594.118,A -85,B 0,C 180,E1 -25568.671,E2 -25568.671} C_VEL
LIN {X 0,Y 390.21,Z 598.79,A -85,B 0,C 180,E1 -25571.005,E2 -25571.005} C_VEL
LIN {X 0,Y 392.159,Z 603.081,A -85,B 0,C 180,E1 -25572.715,E2 -25572.715} C_VEL
LIN {X 0,Y 391.837,Z 606.197,A -85,B 0,C 180,E1 -25572.76,E2 -25572.76} C_VEL
LIN {X 0,Y 390.818,Z 613.894,A -85,B 0,C 180,E1 -25572.729,E2 -25572.729} C_VEL
LIN {X 0,Y 387.315,Z 634.447,A -85,B 0,C 180,E1 -25572.124,E2 -25572.124} C_VEL
LIN {X 0,Y 386.463,Z 641.052,A -85,B 0,C 180,E1 -25572.109,E2 -25572.109} C_VEL
LIN {X 0,Y 374.352,Z 755.138,A -85,B 0,C 180,E1 -25573.766,E2 -25573.766} C_VEL
LIN {X 0,Y 369.806,Z 781.433,A -85,B 0,C 180,E1 -25574.229,E2 -25574.229} C_VEL
LIN {X 0,Y 364.642,Z 803.159,A -85,B 0,C 180,E1 -25574.695,E2 -25574.695} C_VEL
LIN {X 0,Y 357.252,Z 827.721,A -85,B 0,C 180,E1 -25575.377,E2 -25575.377} C_VEL
LIN {X 0,Y 349.704,Z 848.375,A -85,B 0,C 180,E1 -25576.115,E2 -25576.115} C_VEL
LIN {X 0,Y 340.065,Z 871.066,A -85,B 0,C 180,E1 -25577.138,E2 -25577.138} C_VEL
LIN {X 0,Y 330.129,Z 891.103,A -85,B 0,C 180,E1 -25578.281,E2 -25578.281} C_VEL
LIN {X 0,Y 319.075,Z 910.991,A -85,B 0,C 180,E1 -25579.664,E2 -25579.664} C_VEL
LIN {X 0,Y 306.575,Z 930.754,A -85,B 0,C 180,E1 -25581.384,E2 -25581.384} C_VEL
LIN {X 0,Y 294.806,Z 947.644,A -85,B 0,C 180,E1 -25583.198,E2 -25583.198} C_VEL
LIN {X 0,Y 280.655,Z 966.042,A -85,B 0,C 180,E1 -25585.662,E2 -25585.662} C_VEL
LIN {X 0,Y 268.56,Z 980.417,A -85,B 0,C 180,E1 -25588.068,E2 -25588.068} C_VEL
LIN {X 0,Y 254.895,Z 995.623,A -85,B 0,C 180,E1 -25591.222,E2 -25591.222} C_VEL
LIN {X 0,Y 241.418,Z 1009.375,A -85,B 0,C 180,E1 -25594.909,E2 -25594.909} C_VEL
LIN {X 0,Y 229.038,Z 1021.468,A -85,B 0,C 180,E1 -25599.006,E2 -25599.006} C_VEL
LIN {X 0,Y 216.312,Z 1033.306,A -85,B 0,C 180,E1 -25604.266,E2 -25604.266} C_VEL
LIN {X 0,Y 206.429,Z 1042.423,A -85,B 0,C 180,E1 -25609.529,E2 -25609.529} C_VEL
LIN {X 0,Y 196.902,Z 1051.326,A -85,B 0,C 180,E1 -25616.391,E2 -25616.391} C_VEL
LIN {X 0,Y 190.973,Z 1057.306,A -85,B 0,C 180,E1 -25622.564,E2 -25622.564} C_VEL
LIN {X 0,Y 186.284,Z 1062.888,A -85,B 0,C 180,E1 -25630.562,E2 -25630.562} C_VEL
LIN {X 0,Y 184.518,Z 1065.824,A -85,B 0,C 180,E1 -25636.844,E2 -25636.844} C_VEL
LIN {X 0,Y 184.004,Z 1067.586,A -85,B 0,C 180,E1 -25642.82,E2 -25642.82} C_VEL
LIN {X 0,Y 184.018,Z 1068.291,A -85,B 0,C 180,E1 -25648.131,E2 -25648.131} C_VEL
LIN {X 0,Y 184.009,Z 1068.214,A -85,B 0,C 180,E1 -25652.803,E2 -25652.803} C_VEL
LIN {X 0,Y 184.015,Z 1067.428,A -85,B 0,C 180,E1 -25657.807,E2 -25657.807} C_VEL
LIN {X 0,Y 184.631,Z 1065.561,A -85,B 0,C 180,E1 -25663.785,E2 -25663.785} C_VEL
LIN {X 0,Y 187.108,Z 1061.772,A -85,B 0,C 180,E1 -25671.308,E2 -25671.308} C_VEL
LIN {X 0,Y 191.452,Z 1056.726,A -85,B 0,C 180,E1 -25678.038,E2 -25678.038} C_VEL
LIN {X 0,Y 198.246,Z 1050.014,A -85,B 0,C 180,E1 -25684.746,E2 -25684.746} C_VEL
LIN {X 0,Y 207.292,Z 1041.501,A -85,B 0,C 180,E1 -25690.996,E2 -25690.996} C_VEL
LIN {X 0,Y 217.375,Z 1032.23,A -85,B 0,C 180,E1 -25696.234,E2 -25696.234} C_VEL
LIN {X 0,Y 230.209,Z 1020.171,A -85,B 0,C 180,E1 -25701.427,E2 -25701.427} C_VEL
LIN {X 0,Y 242.053,Z 1008.577,A -85,B 0,C 180,E1 -25705.29,E2 -25705.29} C_VEL
LIN {X 0,Y 256.274,Z 993.881,A -85,B 0,C 180,E1 -25709.133,E2 -25709.133} C_VEL
LIN {X 0,Y 269.367,Z 979.247,A -85,B 0,C 180,E1 -25712.114,E2 -25712.114} C_VEL
LIN {X 0,Y 283.436,Z 962.361,A -85,B 0,C 180,E1 -25714.862,E2 -25714.862} C_VEL
LIN {X 0,Y 296.788,Z 944.552,A -85,B 0,C 180,E1 -25717.136,E2 -25717.136} C_VEL
LIN {X 0,Y 309.856,Z 925.503,A -85,B 0,C 180,E1 -25719.099,E2 -25719.099} C_VEL
LIN {X 0,Y 322.006,Z 905.408,A -85,B 0,C 180,E1 -25720.73,E2 -25720.73} C_VEL
LIN {X 0,Y 333.121,Z 884.942,A -85,B 0,C 180,E1 -25722.082,E2 -25722.082} C_VEL
LIN {X 0,Y 343.104,Z 863.625,A -85,B 0,C 180,E1 -25723.202,E2 -25723.202} C_VEL
LIN {X 0,Y 351.013,Z 844.336,A -85,B 0,C 180,E1 -25724.027,E2 -25724.027} C_VEL
LIN {X 0,Y 359.682,Z 819.327,A -85,B 0,C 180,E1 -25724.868,E2 -25724.868} C_VEL
LIN {X 0,Y 365.805,Z 797.571,A -85,B 0,C 180,E1 -25725.425,E2 -25725.425} C_VEL
LIN {X 0,Y 371.457,Z 771.607,A -85,B 0,C 180,E1 -25725.943,E2 -25725.943} C_VEL
LIN {X 0,Y 374.831,Z 749.052,A -85,B 0,C 180,E1 -25726.317,E2 -25726.317} C_VEL
LIN {X 0,Y 389.568,Z 608.29,A -85,B 0,C 180,E1 -25728.376,E2 -25728.376} C_VEL
LIN {X 0,Y 386.964,Z 602.648,A -85,B 0,C 180,E1 -25731.006,E2 -25731.006} C_VEL
LIN {X 0,Y 385.634,Z 599.838,A -85,B 0,C 180,E1 -25732.701,E2 -25732.701} C_VEL
LIN {X 0,Y 384.328,Z 596.847,A -85,B 0,C 180,E1 -25734.925,E2 -25734.925} C_VEL
LIN {X 0,Y 383.162,Z 593.035,A -85,B 0,C 180,E1 -25740.299,E2 -25740.299} C_VEL
LIN {X 0,Y 384.608,Z 597.477,A -85,B 0,C 180,E1 -25746.044,E2 -25746.044} C_VEL
LIN {X 0,Y 386.495,Z 601.651,A -85,B 0,C 180,E1 -25748.855,E2 -25748.855} C_VEL
LIN {X 0,Y 388.896,Z 606.742,A -85,B 0,C 180,E1 -25751.419,E2 -25751.419} C_VEL
LIN {X 0,Y 389.526,Z 608.412,A -85,B 0,C 180,E1 -25752.025,E2 -25752.025} C_VEL
LIN {X 0,Y 374.523,Z 749.949,A -85,B 0,C 180,E1 -25754.067,E2 -25754.067} C_VEL
LIN {X 0,Y 370.042,Z 776.176,A -85,B 0,C 180,E1 -25754.544,E2 -25754.544} C_VEL
LIN {X 0,Y 365.066,Z 797.467,A -85,B 0,C 180,E1 -25755.044,E2 -25755.044} C_VEL
LIN {X 0,Y 357.52,Z 822.95,A -85,B 0,C 180,E1 -25755.83,E2 -25755.83} C_VEL
LIN {X 0,Y 350.119,Z 843.431,A -85,B 0,C 180,E1 -25756.637,E2 -25756.637} C_VEL
LIN {X 0,Y 340.645,Z 865.881,A -85,B 0,C 180,E1 -25757.731,E2 -25757.731} C_VEL
LIN {X 0,Y 330.849,Z 885.699,A -85,B 0,C 180,E1 -25758.925,E2 -25758.925} C_VEL
LIN {X 0,Y 319.956,Z 905.353,A -85,B 0,C 180,E1 -25760.361,E2 -25760.361} C_VEL
LIN {X 0,Y 307.483,Z 925.087,A -85,B 0,C 180,E1 -25762.161,E2 -25762.161} C_VEL
LIN {X 0,Y 295.245,Z 942.592,A -85,B 0,C 180,E1 -25764.119,E2 -25764.119} C_VEL
LIN {X 0,Y 281.522,Z 960.229,A -85,B 0,C 180,E1 -25766.585,E2 -25766.585} C_VEL
LIN {X 0,Y 269.029,Z 974.935,A -85,B 0,C 180,E1 -25769.142,E2 -25769.142} C_VEL
LIN {X 0,Y 254.206,Z 990.991,A -85,B 0,C 180,E1 -25772.676,E2 -25772.676} C_VEL
LIN {X 0,Y 242.305,Z 1002.93,A -85,B 0,C 180,E1 -25776.021,E2 -25776.021} C_VEL
LIN {X 0,Y 228.932,Z 1015.652,A -85,B 0,C 180,E1 -25780.539,E2 -25780.539} C_VEL
LIN {X 0,Y 217.542,Z 1025.868,A -85,B 0,C 180,E1 -25785.313,E2 -25785.313} C_VEL
LIN {X 0,Y 206.816,Z 1035.4,A -85,B 0,C 180,E1 -25791.06,E2 -25791.06} C_VEL
LIN {X 0,Y 198.108,Z 1042.996,A -85,B 0,C 180,E1 -25797.313,E2 -25797.313} C_VEL
LIN {X 0,Y 191.582,Z 1049.113,A -85,B 0,C 180,E1 -25803.998,E2 -25803.998} C_VEL
LIN {X 0,Y 187.096,Z 1053.731,A -85,B 0,C 180,E1 -25811.298,E2 -25811.298} C_VEL
LIN {X 0,Y 184.973,Z 1056.501,A -85,B 0,C 180,E1 -25817.83,E2 -25817.83} C_VEL
LIN {X 0,Y 184.145,Z 1058.203,A -85,B 0,C 180,E1 -25824.704,E2 -25824.704} C_VEL
LIN {X 0,Y 184.042,Z 1058.542,A -85,B 0,C 180,E1 -25830.934,E2 -25830.934} C_VEL
LIN {X 0,Y 184.234,Z 1057.909,A -85,B 0,C 180,E1 -25836.858,E2 -25836.858} C_VEL
LIN {X 0,Y 185.092,Z 1056.34,A -85,B 0,C 180,E1 -25842.797,E2 -25842.797} C_VEL
LIN {X 0,Y 187.346,Z 1053.503,A -85,B 0,C 180,E1 -25849.324,E2 -25849.324} C_VEL
LIN {X 0,Y 192.496,Z 1048.247,A -85,B 0,C 180,E1 -25857.2,E2 -25857.2} C_VEL
LIN {X 0,Y 198.702,Z 1042.554,A -85,B 0,C 180,E1 -25863.264,E2 -25863.264} C_VEL
LIN {X 0,Y 208.439,Z 1034.019,A -85,B 0,C 180,E1 -25870.001,E2 -25870.001} C_VEL
LIN {X 0,Y 218.452,Z 1025.184,A -85,B 0,C 180,E1 -25875.191,E2 -25875.191} C_VEL
LIN {X 0,Y 231.139,Z 1013.75,A -85,B 0,C 180,E1 -25880.356,E2 -25880.356} C_VEL
LIN {X 0,Y 243.459,Z 1001.975,A -85,B 0,C 180,E1 -25884.409,E2 -25884.409} C_VEL
LIN {X 0,Y 256.83,Z 988.547,A -85,B 0,C 180,E1 -25888.073,E2 -25888.073} C_VEL
LIN {X 0,Y 270.716,Z 973.243,A -85,B 0,C 180,E1 -25891.304,E2 -25891.304} C_VEL
LIN {X 0,Y 283.844,Z 957.707,A -85,B 0,C 180,E1 -25893.933,E2 -25893.933} C_VEL
LIN {X 0,Y 297.289,Z 940.068,A -85,B 0,C 180,E1 -25896.303,E2 -25896.303} C_VEL
LIN {X 0,Y 309.145,Z 922.984,A -85,B 0,C 180,E1 -25898.166,E2 -25898.166} C_VEL
LIN {X 0,Y 322.321,Z 901.641,A -85,B 0,C 180,E1 -25900.044,E2 -25900.044} C_VEL
LIN {X 0,Y 332.428,Z 883.2,A -85,B 0,C 180,E1 -25901.347,E2 -25901.347} C_VEL
LIN {X 0,Y 343.533,Z 859.971,A -85,B 0,C 180,E1 -25902.685,E2 -25902.685} C_VEL
LIN {X 0,Y 351.312,Z 841.045,A -85,B 0,C 180,E1 -25903.568,E2 -25903.568} C_VEL
LIN {X 0,Y 359.608,Z 817.534,A -85,B 0,C 180,E1 -25904.46,E2 -25904.46} C_VEL
LIN {X 0,Y 366.16,Z 794.26,A -85,B 0,C 180,E1 -25905.143,E2 -25905.143} C_VEL
LIN {X 0,Y 371.593,Z 770.05,A -85,B 0,C 180,E1 -25905.688,E2 -25905.688} C_VEL
LIN {X 0,Y 375.329,Z 745.784,A -85,B 0,C 180,E1 -25906.098,E2 -25906.098} C_VEL
LIN {X 0,Y 389.812,Z 608.447,A -85,B 0,C 180,E1 -25908.076,E2 -25908.076} C_VEL
LIN {X 0,Y 387.47,Z 603.419,A -85,B 0,C 180,E1 -25910.419,E2 -25910.419} C_VEL
LIN {X 0,Y 385.897,Z 600.084,A -85,B 0,C 180,E1 -25912.406,E2 -25912.406} C_VEL
LIN {X 0,Y 384.54,Z 596.948,A -85,B 0,C 180,E1 -25914.778,E2 -25914.778} C_VEL
LIN {X 0,Y 383.439,Z 593.738,A -85,B 0,C 180,E1 -25920,E2 -25920} C_VEL
LIN {X 0,Y 384.855,Z 597.594,A -85,B 0,C 180,E1 -25925.516,E2 -25925.516} C_VEL
LIN {X 0,Y 386.76,Z 601.807,A -85,B 0,C 180,E1 -25928.399,E2 -25928.399} C_VEL
LIN {X 0,Y 388.975,Z 606.643,A -85,B 0,C 180,E1 -25930.816,E2 -25930.816} C_VEL
LIN {X 0,Y 389.849,Z 608.781,A -85,B 0,C 180,E1 -25931.649,E2 -25931.649} C_VEL
LIN {X 0,Y 386.463,Z 641.052,A -85,B 0,C 180,E1 -25932.109,E2 -25932.109} C_VEL
LIN {X 0,Y 385.442,Z 648.749,A -85,B 0,C 180,E1 -25932.072,E2 -25932.072} C_VEL
LIN {X 0,Y 381.977,Z 669.294,A -85,B 0,C 180,E1 -25931.445,E2 -25931.445} C_VEL
LIN {X 0,Y 381.131,Z 675.896,A -85,B 0,C 180,E1 -25931.432,E2 -25931.432} C_VEL
LIN {X 0,Y 372.424,Z 755.721,A -85,B 0,C 180,E1 -25932.578,E2 -25932.578} C_VEL
LIN {X 0,Y 367.852,Z 781.519,A -85,B 0,C 180,E1 -25933.022,E2 -25933.022} C_VEL
LIN {X 0,Y 362.592,Z 803.315,A -85,B 0,C 180,E1 -25933.475,E2 -25933.475} C_VEL
LIN {X 0,Y 355.199,Z 827.513,A -85,B 0,C 180,E1 -25934.123,E2 -25934.123} C_VEL
LIN {X 0,Y 347.551,Z 848.167,A -85,B 0,C 180,E1 -25934.836,E2 -25934.836} C_VEL
LIN {X 0,Y 337.769,Z 870.856,A -85,B 0,C 180,E1 -25935.826,E2 -25935.826} C_VEL
LIN {X 0,Y 327.612,Z 891.006,A -85,B 0,C 180,E1 -25936.941,E2 -25936.941} C_VEL
LIN {X 0,Y 316.429,Z 910.779,A -85,B 0,C 180,E1 -25938.276,E2 -25938.276} C_VEL
LIN {X 0,Y 303.69,Z 930.539,A -85,B 0,C 180,E1 -25939.948,E2 -25939.948} C_VEL
LIN {X 0,Y 291.522,Z 947.639,A -85,B 0,C 180,E1 -25941.742,E2 -25941.742} C_VEL
LIN {X 0,Y 276.404,Z 966.759,A -85,B 0,C 180,E1 -25944.271,E2 -25944.271} C_VEL
LIN {X 0,Y 264.024,Z 981.053,A -85,B 0,C 180,E1 -25946.65,E2 -25946.65} C_VEL
LIN {X 0,Y 249.273,Z 996.827,A -85,B 0,C 180,E1 -25949.954,E2 -25949.954} C_VEL
LIN {X 0,Y 236.108,Z 1009.799,A -85,B 0,C 180,E1 -25953.459,E2 -25953.459} C_VEL
LIN {X 0,Y 222.693,Z 1022.406,A -85,B 0,C 180,E1 -25957.792,E2 -25957.792} C_VEL
LIN {X 0,Y 210.055,Z 1033.564,A -85,B 0,C 180,E1 -25962.899,E2 -25962.899} C_VEL
LIN {X 0,Y 198.84,Z 1043.44,A -85,B 0,C 180,E1 -25968.795,E2 -25968.795} C_VEL
LIN {X 0,Y 189.717,Z 1051.416,A -85,B 0,C 180,E1 -25975.305,E2 -25975.305} C_VEL
LIN {X 0,Y 183.19,Z 1057.609,A -85,B 0,C 180,E1 -25982.004,E2 -25982.004} C_VEL
LIN {X 0,Y 178.443,Z 1062.836,A -85,B 0,C 180,E1 -25990.013,E2 -25990.013} C_VEL
LIN {X 0,Y 176.552,Z 1065.725,A -85,B 0,C 180,E1 -25996.573,E2 -25996.573} C_VEL
LIN {X 0,Y 176.006,Z 1067.442,A -85,B 0,C 180,E1 -26002.82,E2 -26002.82} C_VEL
LIN {X 0,Y 176.027,Z 1068.124,A -85,B 0,C 180,E1 -26008.698,E2 -26008.698} C_VEL
LIN {X 0,Y 175.993,Z 1067.902,A -85,B 0,C 180,E1 -26014.235,E2 -26014.235} C_VEL
LIN {X 0,Y 176.215,Z 1066.573,A -85,B 0,C 180,E1 -26020.993,E2 -26020.993} C_VEL
LIN {X 0,Y 177.823,Z 1063.626,A -85,B 0,C 180,E1 -26028.354,E2 -26028.354} C_VEL
LIN {X 0,Y 181.157,Z 1059.637,A -85,B 0,C 180,E1 -26035.15,E2 -26035.15} C_VEL
LIN {X 0,Y 188.03,Z 1052.895,A -85,B 0,C 180,E1 -26043.211,E2 -26043.211} C_VEL
LIN {X 0,Y 195.817,Z 1045.904,A -85,B 0,C 180,E1 -26049.284,E2 -26049.284} C_VEL
LIN {X 0,Y 206.97,Z 1036.205,A -85,B 0,C 180,E1 -26055.643,E2 -26055.643} C_VEL
LIN {X 0,Y 218.498,Z 1025.952,A -85,B 0,C 180,E1 -26060.658,E2 -26060.658} C_VEL
LIN {X 0,Y 232.131,Z 1013.499,A -85,B 0,C 180,E1 -26065.358,E2 -26065.358} C_VEL
LIN {X 0,Y 245.703,Z 1000.189,A -85,B 0,C 180,E1 -26069.166,E2 -26069.166} C_VEL
LIN {X 0,Y 260.075,Z 985.273,A -85,B 0,C 180,E1 -26072.525,E2 -26072.525} C_VEL
LIN {X 0,Y 274.032,Z 969.313,A -85,B 0,C 180,E1 -26075.306,E2 -26075.306} C_VEL
LIN {X 0,Y 286.777,Z 953.578,A -85,B 0,C 180,E1 -26077.512,E2 -26077.512} C_VEL
LIN {X 0,Y 300.747,Z 934.486,A -85,B 0,C 180,E1 -26079.646,E2 -26079.646} C_VEL
LIN {X 0,Y 312.124,Z 917.225,A -85,B 0,C 180,E1 -26081.197,E2 -26081.197} C_VEL
LIN {X 0,Y 324.607,Z 896.131,A -85,B 0,C 180,E1 -26082.725,E2 -26082.725} C_VEL
LIN {X 0,Y 334.776,Z 876.42,A -85,B 0,C 180,E1 -26083.873,E2 -26083.873} C_VEL
LIN {X 0,Y 344.859,Z 854.309,A -85,B 0,C 180,E1 -26084.907,E2 -26084.907} C_VEL
LIN {X 0,Y 353.38,Z 831.919,A -85,B 0,C 180,E1 -26085.72,E2 -26085.72} C_VEL
LIN {X 0,Y 360.169,Z 810.948,A -85,B 0,C 180,E1 -26086.326,E2 -26086.326} C_VEL
LIN {X 0,Y 366.646,Z 785.75,A -85,B 0,C 180,E1 -26086.887,E2 -26086.887} C_VEL
LIN {X 0,Y 370.932,Z 763.567,A -85,B 0,C 180,E1 -26087.284,E2 -26087.284} C_VEL
LIN {X 0,Y 375.036,Z 730.827,A -85,B 0,C 180,E1 -26087.779,E2 -26087.779} C_VEL
LIN {X 0,Y 387.397,Z 614.116,A -85,B 0,C 180,E1 -26089.441,E2 -26089.441} C_VEL
LIN {X 0,Y 384.927,Z 608.397,A -85,B 0,C 180,E1 -26092.312,E2 -26092.312} C_VEL
LIN {X 0,Y 383.273,Z 604.729,A -85,B 0,C 180,E1 -26095.061,E2 -26095.061} C_VEL
LIN {X 0,Y 382.179,Z 601.043,A -85,B 0,C 180,E1 -26100.3,E2 -26100.3} C_VEL
LIN {X 0,Y 383.505,Z 605.284,A -85,B 0,C 180,E1 -26105.836,E2 -26105.836} C_VEL
LIN {X 0,Y 385.321,Z 609.483,A -85,B 0,C 180,E1 -26108.656,E2 -26108.656} C_VEL
LIN {X 0,Y 387.364,Z 613.986,A -85,B 0,C 180,E1 -26110.942,E2 -26110.942} C_VEL
LIN {X 0,Y 372.645,Z 750.291,A -85,B 0,C 180,E1 -26112.875,E2 -26112.875} C_VEL
LIN {X 0,Y 368.102,Z 776.45,A -85,B 0,C 180,E1 -26113.338,E2 -26113.338} C_VEL
LIN {X 0,Y 363.04,Z 797.8,A -85,B 0,C 180,E1 -26113.825,E2 -26113.825} C_VEL
LIN {X 0,Y 355.414,Z 823.173,A -85,B 0,C 180,E1 -26114.585,E2 -26114.585} C_VEL
LIN {X 0,Y 347.903,Z 843.652,A -85,B 0,C 180,E1 -26115.369,E2 -26115.369} C_VEL
LIN {X 0,Y 338.28,Z 866.101,A -85,B 0,C 180,E1 -26116.432,E2 -26116.432} C_VEL
LIN {X 0,Y 328.32,Z 885.919,A -85,B 0,C 180,E1 -26117.592,E2 -26117.592} C_VEL
LIN {X 0,Y 316.81,Z 906.303,A -85,B 0,C 180,E1 -26119.046,E2 -26119.046} C_VEL
LIN {X 0,Y 304.197,Z 925.771,A -85,B 0,C 180,E1 -26120.793,E2 -26120.793} C_VEL
LIN {X 0,Y 291.612,Z 943.364,A -85,B 0,C 180,E1 -26122.728,E2 -26122.728} C_VEL
LIN {X 0,Y 277.355,Z 961.171,A -85,B 0,C 180,E1 -26125.194,E2 -26125.194} C_VEL
LIN {X 0,Y 264.398,Z 975.993,A -85,B 0,C 180,E1 -26127.757,E2 -26127.757} C_VEL
LIN {X 0,Y 249.172,Z 991.905,A -85,B 0,C 180,E1 -26131.27,E2 -26131.27} C_VEL
LIN {X 0,Y 236.911,Z 1003.779,A -85,B 0,C 180,E1 -26134.614,E2 -26134.614} C_VEL
LIN {X 0,Y 222.48,Z 1016.888,A -85,B 0,C 180,E1 -26139.375,E2 -26139.375} C_VEL
LIN {X 0,Y 211.245,Z 1026.541,A -85,B 0,C 180,E1 -26143.99,E2 -26143.99} C_VEL
LIN {X 0,Y 199.91,Z 1036.074,A -85,B 0,C 180,E1 -26149.931,E2 -26149.931} C_VEL
LIN {X 0,Y 190.903,Z 1043.512,A -85,B 0,C 180,E1 -26156.276,E2 -26156.276} C_VEL
LIN {X 0,Y 183.77,Z 1049.811,A -85,B 0,C 180,E1 -26163.503,E2 -26163.503} C_VEL
LIN {X 0,Y 179.26,Z 1054.104,A -85,B 0,C 180,E1 -26170.786,E2 -26170.786} C_VEL
LIN {X 0,Y 177.079,Z 1056.717,A -85,B 0,C 180,E1 -26177.279,E2 -26177.279} C_VEL
LIN {X 0,Y 176.159,Z 1058.417,A -85,B 0,C 180,E1 -26184.463,E2 -26184.463} C_VEL
LIN {X 0,Y 176.045,Z 1058.755,A -85,B 0,C 180,E1 -26190.977,E2 -26190.977} C_VEL
LIN {X 0,Y 176.259,Z 1058.123,A -85,B 0,C 180,E1 -26197.17,E2 -26197.17} C_VEL
LIN {X 0,Y 177.214,Z 1056.556,A -85,B 0,C 180,E1 -26203.376,E2 -26203.376} C_VEL
LIN {X 0,Y 179.683,Z 1053.72,A -85,B 0,C 180,E1 -26210.183,E2 -26210.183} C_VEL
LIN {X 0,Y 185.299,Z 1048.422,A -85,B 0,C 180,E1 -26218.41,E2 -26218.41} C_VEL
LIN {X 0,Y 191.892,Z 1042.772,A -85,B 0,C 180,E1 -26224.609,E2 -26224.609} C_VEL
LIN {X 0,Y 202.211,Z 1034.237,A -85,B 0,C 180,E1 -26231.499,E2 -26231.499} C_VEL
LIN {X 0,Y 212.734,Z 1025.402,A -85,B 0,C 180,E1 -26236.764,E2 -26236.764} C_VEL
LIN {X 0,Y 225.985,Z 1013.967,A -85,B 0,C 180,E1 -26241.96,E2 -26241.96} C_VEL
LIN {X 0,Y 238.774,Z 1002.192,A -85,B 0,C 180,E1 -26246.011,E2 -26246.011} C_VEL
LIN {X 0,Y 252.591,Z 988.764,A -85,B 0,C 180,E1 -26249.651,E2 -26249.651} C_VEL
LIN {X 0,Y 266.516,Z 973.871,A -85,B 0,C 180,E1 -26252.767,E2 -26252.767} C_VEL
LIN {X 0,Y 279.571,Z 958.839,A -85,B 0,C 180,E1 -26255.29,E2 -26255.29} C_VEL
LIN {X 0,Y 293.911,Z 940.559,A -85,B 0,C 180,E1 -26257.721,E2 -26257.721} C_VEL
LIN {X 0,Y 305.867,Z 923.71,A -85,B 0,C 180,E1 -26259.526,E2 -26259.526} C_VEL
LIN {X 0,Y 319.449,Z 902.198,A -85,B 0,C 180,E1 -26261.381,E2 -26261.381} C_VEL
LIN {X 0,Y 329.502,Z 884.218,A -85,B 0,C 180,E1 -26262.624,E2 -26262.624} C_VEL
LIN {X 0,Y 340.352,Z 862.181,A -85,B 0,C 180,E1 -26263.877,E2 -26263.877} C_VEL
LIN {X 0,Y 349.124,Z 841.252,A -85,B 0,C 180,E1 -26264.833,E2 -26264.833} C_VEL
LIN {X 0,Y 357.32,Z 818.473,A -85,B 0,C 180,E1 -26265.676,E2 -26265.676} C_VEL
LIN {X 0,Y 364.125,Z 794.702,A -85,B 0,C 180,E1 -26266.356,E2 -26266.356} C_VEL
LIN {X 0,Y 369.663,Z 770.435,A -85,B 0,C 180,E1 -26266.887,E2 -26266.887} C_VEL
LIN {X 0,Y 373.473,Z 746.083,A -85,B 0,C 180,E1 -26267.289,E2 -26267.289} C_VEL
LIN {X 0,Y 387.61,Z 614.147,A -85,B 0,C 180,E1 -26269.183,E2 -26269.183} C_VEL
LIN {X 0,Y 385.134,Z 608.528,A -85,B 0,C 180,E1 -26272.091,E2 -26272.091} C_VEL
LIN {X 0,Y 383.489,Z 604.832,A -85,B 0,C 180,E1 -26274.914,E2 -26274.914} C_VEL
LIN {X 0,Y 382.459,Z 601.718,A -85,B 0,C 180,E1 -26280,E2 -26280} C_VEL
LIN {X 0,Y 383.79,Z 605.508,A -85,B 0,C 180,E1 -26285.382,E2 -26285.382} C_VEL
LIN {X 0,Y 385.588,Z 609.634,A -85,B 0,C 180,E1 -26288.2,E2 -26288.2} C_VEL
LIN {X 0,Y 387.687,Z 614.375,A -85,B 0,C 180,E1 -26290.568,E2 -26290.568} C_VEL
LIN {X 0,Y 381.131,Z 675.896,A -85,B 0,C 180,E1 -26291.432,E2 -26291.432} C_VEL
LIN {X 0,Y 380.118,Z 683.591,A -85,B 0,C 180,E1 -26291.396,E2 -26291.396} C_VEL
LIN {X 0,Y 376.697,Z 704.129,A -85,B 0,C 180,E1 -26290.748,E2 -26290.748} C_VEL
LIN {X 0,Y 375.847,Z 710.733,A -85,B 0,C 180,E1 -26290.729,E2 -26290.729} C_VEL
LIN {X 0,Y 370.348,Z 758.675,A -85,B 0,C 180,E1 -26291.414,E2 -26291.414} C_VEL
LIN {X 0,Y 365.694,Z 783.281,A -85,B 0,C 180,E1 -26291.833,E2 -26291.833} C_VEL
LIN {X 0,Y 359.751,Z 807.104,A -85,B 0,C 180,E1 -26292.323,E2 -26292.323} C_VEL
LIN {X 0,Y 352.406,Z 829.883,A -85,B 0,C 180,E1 -26292.936,E2 -26292.936} C_VEL
LIN {X 0,Y 344.214,Z 851.359,A -85,B 0,C 180,E1 -26293.67,E2 -26293.67} C_VEL
LIN {X 0,Y 333.854,Z 874.261,A -85,B 0,C 180,E1 -26294.674,E2 -26294.674} C_VEL
LIN {X 0,Y 324.074,Z 893.126,A -85,B 0,C 180,E1 -26295.711,E2 -26295.711} C_VEL
LIN {X 0,Y 310.918,Z 915.378,A -85,B 0,C 180,E1 -26297.228,E2 -26297.228} C_VEL
LIN {X 0,Y 299.427,Z 932.584,A -85,B 0,C 180,E1 -26298.698,E2 -26298.698} C_VEL
LIN {X 0,Y 285.42,Z 951.595,A -85,B 0,C 180,E1 -26300.713,E2 -26300.713} C_VEL
LIN {X 0,Y 271.518,Z 968.41,A -85,B 0,C 180,E1 -26302.979,E2 -26302.979} C_VEL
LIN {X 0,Y 257.339,Z 984.249,A -85,B 0,C 180,E1 -26305.652,E2 -26305.652} C_VEL
LIN {X 0,Y 242.316,Z 999.442,A -85,B 0,C 180,E1 -26308.979,E2 -26308.979} C_VEL
LIN {X 0,Y 228.899,Z 1012.151,A -85,B 0,C 180,E1 -26312.534,E2 -26312.534} C_VEL
LIN {X 0,Y 214.576,Z 1024.809,A -85,B 0,C 180,E1 -26317.171,E2 -26317.171} C_VEL
LIN {X 0,Y 202.893,Z 1034.695,A -85,B 0,C 180,E1 -26321.913,E2 -26321.913} C_VEL
LIN {X 0,Y 190.368,Z 1045.048,A -85,B 0,C 180,E1 -26328.562,E2 -26328.562} C_VEL
LIN {X 0,Y 181.878,Z 1052.127,A -85,B 0,C 180,E1 -26334.743,E2 -26334.743} C_VEL
LIN {X 0,Y 174.432,Z 1058.826,A -85,B 0,C 180,E1 -26342.704,E2 -26342.704} C_VEL
LIN {X 0,Y 170.341,Z 1063.114,A -85,B 0,C 180,E1 -26350.095,E2 -26350.095} C_VEL
LIN {X 0,Y 168.421,Z 1065.982,A -85,B 0,C 180,E1 -26357.31,E2 -26357.31} C_VEL
LIN {X 0,Y 167.992,Z 1067.618,A -85,B 0,C 180,E1 -26364.535,E2 -26364.535} C_VEL
LIN {X 0,Y 168.039,Z 1067.975,A -85,B 0,C 180,E1 -26370.341,E2 -26370.341} C_VEL
LIN {X 0,Y 167.992,Z 1067.425,A -85,B 0,C 180,E1 -26376.493,E2 -26376.493} C_VEL
LIN {X 0,Y 168.531,Z 1065.719,A -85,B 0,C 180,E1 -26383.378,E2 -26383.378} C_VEL
LIN {X 0,Y 170.475,Z 1062.911,A -85,B 0,C 180,E1 -26390.246,E2 -26390.246} C_VEL
LIN {X 0,Y 175.168,Z 1058.113,A -85,B 0,C 180,E1 -26398.279,E2 -26398.279} C_VEL
LIN {X 0,Y 182.58,Z 1051.448,A -85,B 0,C 180,E1 -26405.853,E2 -26405.853} C_VEL
LIN {X 0,Y 192.2,Z 1043.516,A -85,B 0,C 180,E1 -26412.555,E2 -26412.555} C_VEL
LIN {X 0,Y 203.987,Z 1033.65,A -85,B 0,C 180,E1 -26418.587,E2 -26418.587} C_VEL
LIN {X 0,Y 217.067,Z 1022.593,A -85,B 0,C 180,E1 -26423.718,E2 -26423.718} C_VEL
LIN {X 0,Y 231.367,Z 1009.662,A -85,B 0,C 180,E1 -26428.181,E2 -26428.181} C_VEL
LIN {X 0,Y 245.687,Z 995.991,A -85,B 0,C 180,E1 -26431.83,E2 -26431.83} C_VEL
LIN {X 0,Y 260.812,Z 980.169,A -85,B 0,C 180,E1 -26435.057,E2 -26435.057} C_VEL
LIN {X 0,Y 274.727,Z 964.422,A -85,B 0,C 180,E1 -26437.585,E2 -26437.585} C_VEL
LIN {X 0,Y 289.559,Z 945.785,A -85,B 0,C 180,E1 -26439.926,E2 -26439.926} C_VEL
LIN {X 0,Y 302.133,Z 928.329,A -85,B 0,C 180,E1 -26441.676,E2 -26441.676} C_VEL
LIN {X 0,Y 315.637,Z 907.282,A -85,B 0,C 180,E1 -26443.347,E2 -26443.347} C_VEL
LIN {X 0,Y 326.209,Z 888.685,A -85,B 0,C 180,E1 -26444.534,E2 -26444.534} C_VEL
LIN {X 0,Y 337.434,Z 866.207,A -85,B 0,C 180,E1 -26445.689,E2 -26445.689} C_VEL
LIN {X 0,Y 346.01,Z 846.16,A -85,B 0,C 180,E1 -26446.509,E2 -26446.509} C_VEL
LIN {X 0,Y 354.676,Z 822.587,A -85,B 0,C 180,E1 -26447.273,E2 -26447.273} C_VEL
LIN {X 0,Y 361.566,Z 799.116,A -85,B 0,C 180,E1 -26447.845,E2 -26447.845} C_VEL
LIN {X 0,Y 367.262,Z 774.725,A -85,B 0,C 180,E1 -26448.312,E2 -26448.312} C_VEL
LIN {X 0,Y 371.133,Z 750.319,A -85,B 0,C 180,E1 -26448.701,E2 -26448.701} C_VEL
LIN {X 0,Y 385.321,Z 619.987,A -85,B 0,C 180,E1 -26450.546,E2 -26450.546} C_VEL
LIN {X 0,Y 383.453,Z 615.629,A -85,B 0,C 180,E1 -26452.96,E2 -26452.96} C_VEL
LIN {X 0,Y 382.145,Z 612.518,A -85,B 0,C 180,E1 -26455.347,E2 -26455.347} C_VEL
LIN {X 0,Y 381.196,Z 609.049,A -85,B 0,C 180,E1 -26460.301,E2 -26460.301} C_VEL
LIN {X 0,Y 382.441,Z 613.204,A -85,B 0,C 180,E1 -26465.702,E2 -26465.702} C_VEL
LIN {X 0,Y 384.153,Z 617.313,A -85,B 0,C 180,E1 -26468.457,E2 -26468.457} C_VEL
LIN {X 0,Y 385.285,Z 620.101,A -85,B 0,C 180,E1 -26469.856,E2 -26469.856} C_VEL
LIN {X 0,Y 370.944,Z 750.526,A -85,B 0,C 180,E1 -26471.67,E2 -26471.67} C_VEL
LIN {X 0,Y 366.335,Z 776.69,A -85,B 0,C 180,E1 -26472.12,E2 -26472.12} C_VEL
LIN {X 0,Y 361.181,Z 798.134,A -85,B 0,C 180,E1 -26472.593,E2 -26472.593} C_VEL
LIN {X 0,Y 353.478,Z 823.395,A -85,B 0,C 180,E1 -26473.326,E2 -26473.326} C_VEL
LIN {X 0,Y 345.86,Z 843.874,A -85,B 0,C 180,E1 -26474.085,E2 -26474.085} C_VEL
LIN {X 0,Y 336.217,Z 866.065,A -85,B 0,C 180,E1 -26475.101,E2 -26475.101} C_VEL
LIN {X 0,Y 325.971,Z 886.14,A -85,B 0,C 180,E1 -26476.24,E2 -26476.24} C_VEL
LIN {X 0,Y 314.261,Z 906.524,A -85,B 0,C 180,E1 -26477.651,E2 -26477.651} C_VEL
LIN {X 0,Y 301.439,Z 925.95,A -85,B 0,C 180,E1 -26479.347,E2 -26479.347} C_VEL
LIN {X 0,Y 288.566,Z 943.585,A -85,B 0,C 180,E1 -26481.237,E2 -26481.237} C_VEL
LIN {X 0,Y 273.981,Z 961.392,A -85,B 0,C 180,E1 -26483.65,E2 -26483.65} C_VEL
LIN {X 0,Y 260.619,Z 976.292,A -85,B 0,C 180,E1 -26486.181,E2 -26486.181} C_VEL
LIN {X 0,Y 245.019,Z 992.126,A -85,B 0,C 180,E1 -26489.632,E2 -26489.632} C_VEL
LIN {X 0,Y 232.346,Z 1004,A -85,B 0,C 180,E1 -26492.948,E2 -26492.948} C_VEL
LIN {X 0,Y 217.221,Z 1017.223,A -85,B 0,C 180,E1 -26497.75,E2 -26497.75} C_VEL
LIN {X 0,Y 205.618,Z 1026.761,A -85,B 0,C 180,E1 -26502.341,E2 -26502.341} C_VEL
LIN {X 0,Y 193.835,Z 1036.191,A -85,B 0,C 180,E1 -26508.284,E2 -26508.284} C_VEL
LIN {X 0,Y 184.135,Z 1043.732,A -85,B 0,C 180,E1 -26514.859,E2 -26514.859} C_VEL
LIN {X 0,Y 176.489,Z 1050.03,A -85,B 0,C 180,E1 -26522.318,E2 -26522.318} C_VEL
LIN {X 0,Y 171.6,Z 1054.321,A -85,B 0,C 180,E1 -26529.893,E2 -26529.893} C_VEL
LIN {X 0,Y 169.124,Z 1057.043,A -85,B 0,C 180,E1 -26537.017,E2 -26537.017} C_VEL
LIN {X 0,Y 168.157,Z 1058.678,A -85,B 0,C 180,E1 -26544.541,E2 -26544.541} C_VEL
LIN {X 0,Y 168.048,Z 1058.968,A -85,B 0,C 180,E1 -26551.023,E2 -26551.023} C_VEL
LIN {X 0,Y 168.289,Z 1058.337,A -85,B 0,C 180,E1 -26557.511,E2 -26557.511} C_VEL
LIN {X 0,Y 169.351,Z 1056.771,A -85,B 0,C 180,E1 -26564.009,E2 -26564.009} C_VEL
LIN {X 0,Y 172.062,Z 1053.937,A -85,B 0,C 180,E1 -26571.119,E2 -26571.119} C_VEL
LIN {X 0,Y 178.091,Z 1048.682,A -85,B 0,C 180,E1 -26579.609,E2 -26579.609} C_VEL
LIN {X 0,Y 185.191,Z 1042.99,A -85,B 0,C 180,E1 -26586.052,E2 -26586.052} C_VEL
LIN {X 0,Y 196.127,Z 1034.456,A -85,B 0,C 180,E1 -26593.091,E2 -26593.091} C_VEL
LIN {X 0,Y 207.186,Z 1025.62,A -85,B 0,C 180,E1 -26598.421,E2 -26598.421} C_VEL
LIN {X 0,Y 221.016,Z 1014.185,A -85,B 0,C 180,E1 -26603.638,E2 -26603.638} C_VEL
LIN {X 0,Y 234.283,Z 1002.409,A -85,B 0,C 180,E1 -26607.676,E2 -26607.676} C_VEL
LIN {X 0,Y 248.552,Z 988.98,A -85,B 0,C 180,E1 -26611.281,E2 -26611.281} C_VEL
LIN {X 0,Y 262.876,Z 974.087,A -85,B 0,C 180,E1 -26614.352,E2 -26614.352} C_VEL
LIN {X 0,Y 276.261,Z 959.054,A -85,B 0,C 180,E1 -26616.827,E2 -26616.827} C_VEL
LIN {X 0,Y 290.925,Z 940.773,A -85,B 0,C 180,E1 -26619.204,E2 -26619.204} C_VEL
LIN {X 0,Y 302.798,Z 924.388,A -85,B 0,C 180,E1 -26620.918,E2 -26620.918} C_VEL
LIN {X 0,Y 316.698,Z 902.85,A -85,B 0,C 180,E1 -26622.736,E2 -26622.736} C_VEL
LIN {X 0,Y 327.182,Z 884.428,A -85,B 0,C 180,E1 -26623.974,E2 -26623.974} C_VEL
LIN {X 0,Y 338.203,Z 862.39,A -85,B 0,C 180,E1 -26625.188,E2 -26625.188} C_VEL
LIN {X 0,Y 347.108,Z 841.46,A -85,B 0,C 180,E1 -26626.114,E2 -26626.114} C_VEL
LIN {X 0,Y 355.42,Z 818.678,A -85,B 0,C 180,E1 -26626.93,E2 -26626.93} C_VEL
LIN {X 0,Y 362.267,Z 795.1,A -85,B 0,C 180,E1 -26627.583,E2 -26627.583} C_VEL
LIN {X 0,Y 367.872,Z 770.943,A -85,B 0,C 180,E1 -26628.096,E2 -26628.096} C_VEL
LIN {X 0,Y 371.766,Z 746.489,A -85,B 0,C 180,E1 -26628.489,E2 -26628.489} C_VEL
LIN {X 0,Y 385.578,Z 620.099,A -85,B 0,C 180,E1 -26630.254,E2 -26630.254} C_VEL
LIN {X 0,Y 383.62,Z 615.683,A -85,B 0,C 180,E1 -26632.813,E2 -26632.813} C_VEL
LIN {X 0,Y 382.44,Z 612.716,A -85,B 0,C 180,E1 -26635.05,E2 -26635.05} C_VEL
LIN {X 0,Y 381.479,Z 609.697,A -85,B 0,C 180,E1 -26640,E2 -26640} C_VEL
LIN {X 0,Y 382.693,Z 613.311,A -85,B 0,C 180,E1 -26645.172,E2 -26645.172} C_VEL
LIN {X 0,Y 384.421,Z 617.459,A -85,B 0,C 180,E1 -26647.999,E2 -26647.999} C_VEL
LIN {X 0,Y 385.622,Z 620.374,A -85,B 0,C 180,E1 -26649.483,E2 -26649.483} C_VEL
LIN {X 0,Y 375.847,Z 710.733,A -85,B 0,C 180,E1 -26650.729,E2 -26650.729} C_VEL
LIN {X 0,Y 374.856,Z 718.429,A -85,B 0,C 180,E1 -26650.689,E2 -26650.689} C_VEL
LIN {X 0,Y 371.5,Z 738.965,A -85,B 0,C 180,E1 -26650.026,E2 -26650.026} C_VEL
LIN {X 0,Y 370.543,Z 745.555,A -85,B 0,C 180,E1 -26650.003,E2 -26650.003} C_VEL
LIN {X 0,Y 367.124,Z 768.25,A -85,B 0,C 180,E1 -26650.346,E2 -26650.346} C_VEL
LIN {X 0,Y 361.754,Z 793.321,A -85,B 0,C 180,E1 -26650.782,E2 -26650.782} C_VEL
LIN {X 0,Y 355.479,Z 815.357,A -85,B 0,C 180,E1 -26651.267,E2 -26651.267} C_VEL
LIN {X 0,Y 347.927,Z 837.402,A -85,B 0,C 180,E1 -26651.889,E2 -26651.889} C_VEL
LIN {X 0,Y 338.734,Z 859.523,A -85,B 0,C 180,E1 -26652.686,E2 -26652.686} C_VEL
LIN {X 0,Y 329.175,Z 879.475,A -85,B 0,C 180,E1 -26653.585,E2 -26653.585} C_VEL
LIN {X 0,Y 316.595,Z 902.23,A -85,B 0,C 180,E1 -26654.888,E2 -26654.888} C_VEL
LIN {X 0,Y 305.073,Z 920.535,A -85,B 0,C 180,E1 -26656.194,E2 -26656.194} C_VEL
LIN {X 0,Y 290.297,Z 941.411,A -85,B 0,C 180,E1 -26658.076,E2 -26658.076} C_VEL
LIN {X 0,Y 277.559,Z 957.507,A -85,B 0,C 180,E1 -26659.908,E2 -26659.908} C_VEL
LIN {X 0,Y 262.38,Z 974.983,A -85,B 0,C 180,E1 -26662.401,E2 -26662.401} C_VEL
LIN {X 0,Y 247.594,Z 990.31,A -85,B 0,C 180,E1 -26665.229,E2 -26665.229} C_VEL
LIN {X 0,Y 232.479,Z 1004.861,A -85,B 0,C 180,E1 -26668.669,E2 -26668.669} C_VEL
LIN {X 0,Y 217.613,Z 1017.904,A -85,B 0,C 180,E1 -26672.77,E2 -26672.77} C_VEL
LIN {X 0,Y 203.396,Z 1029.804,A -85,B 0,C 180,E1 -26677.676,E2 -26677.676} C_VEL
LIN {X 0,Y 190.793,Z 1039.698,A -85,B 0,C 180,E1 -26683.242,E2 -26683.242} C_VEL
LIN {X 0,Y 180.066,Z 1048.116,A -85,B 0,C 180,E1 -26689.531,E2 -26689.531} C_VEL
LIN {X 0,Y 170.948,Z 1055.342,A -85,B 0,C 180,E1 -26697.046,E2 -26697.046} C_VEL
LIN {X 0,Y 165.246,Z 1060.312,A -85,B 0,C 180,E1 -26704.172,E2 -26704.172} C_VEL
LIN {X 0,Y 161.292,Z 1064.579,A -85,B 0,C 180,E1 -26713.06,E2 -26713.06} C_VEL
LIN {X 0,Y 160.103,Z 1066.654,A -85,B 0,C 180,E1 -26720.292,E2 -26720.292} C_VEL
LIN {X 0,Y 160.004,Z 1067.553,A -85,B 0,C 180,E1 -26726.417,E2 -26726.417} C_VEL
LIN {X 0,Y 160.026,Z 1067.668,A -85,B 0,C 180,E1 -26731.79,E2 -26731.79} C_VEL
LIN {X 0,Y 160.02,Z 1066.996,A -85,B 0,C 180,E1 -26737.901,E2 -26737.901} C_VEL
LIN {X 0,Y 160.774,Z 1065.264,A -85,B 0,C 180,E1 -26744.773,E2 -26744.773} C_VEL
LIN {X 0,Y 163.297,Z 1062.195,A -85,B 0,C 180,E1 -26752.311,E2 -26752.311} C_VEL
LIN {X 0,Y 169.091,Z 1056.842,A -85,B 0,C 180,E1 -26760.97,E2 -26760.97} C_VEL
LIN {X 0,Y 176.346,Z 1050.9,A -85,B 0,C 180,E1 -26767.76,E2 -26767.76} C_VEL
LIN {X 0,Y 187.17,Z 1042.483,A -85,B 0,C 180,E1 -26774.842,E2 -26774.842} C_VEL
LIN {X 0,Y 199.18,Z 1032.96,A -85,B 0,C 180,E1 -26780.631,E2 -26780.631} C_VEL
LIN {X 0,Y 212.925,Z 1021.827,A -85,B 0,C 180,E1 -26785.74,E2 -26785.74} C_VEL
LIN {X 0,Y 227.383,Z 1009.194,A -85,B 0,C 180,E1 -26790.029,E2 -26790.029} C_VEL
LIN {X 0,Y 242.193,Z 995.491,A -85,B 0,C 180,E1 -26793.621,E2 -26793.621} C_VEL
LIN {X 0,Y 257.036,Z 980.384,A -85,B 0,C 180,E1 -26796.643,E2 -26796.643} C_VEL
LIN {X 0,Y 270.872,Z 965.133,A -85,B 0,C 180,E1 -26799.054,E2 -26799.054} C_VEL
LIN {X 0,Y 286.24,Z 946.366,A -85,B 0,C 180,E1 -26801.376,E2 -26801.376} C_VEL
LIN {X 0,Y 298.929,Z 929.142,A -85,B 0,C 180,E1 -26803.066,E2 -26803.066} C_VEL
LIN {X 0,Y 313.018,Z 907.698,A -85,B 0,C 180,E1 -26804.729,E2 -26804.729} C_VEL
LIN {X 0,Y 323.771,Z 889.13,A -85,B 0,C 180,E1 -26805.879,E2 -26805.879} C_VEL
LIN {X 0,Y 335.005,Z 867.14,A -85,B 0,C 180,E1 -26806.978,E2 -26806.978} C_VEL
LIN {X 0,Y 344.217,Z 845.938,A -85,B 0,C 180,E1 -26807.814,E2 -26807.814} C_VEL
LIN {X 0,Y 352.758,Z 823.083,A -85,B 0,C 180,E1 -26808.528,E2 -26808.528} C_VEL
LIN {X 0,Y 359.872,Z 799.216,A -85,B 0,C 180,E1 -26809.089,E2 -26809.089} C_VEL
LIN {X 0,Y 365.633,Z 774.951,A -85,B 0,C 180,E1 -26809.537,E2 -26809.537} C_VEL
LIN {X 0,Y 369.618,Z 750.277,A -85,B 0,C 180,E1 -26809.919,E2 -26809.919} C_VEL
LIN {X 0,Y 383.39,Z 626.045,A -85,B 0,C 180,E1 -26811.64,E2 -26811.64} C_VEL
LIN {X 0,Y 382.077,Z 622.94,A -85,B 0,C 180,E1 -26813.539,E2 -26813.539} C_VEL
LIN {X 0,Y 381.097,Z 620.399,A -85,B 0,C 180,E1 -26815.485,E2 -26815.485} C_VEL
LIN {X 0,Y 380.213,Z 617.052,A -85,B 0,C 180,E1 -26820.301,E2 -26820.301} C_VEL
LIN {X 0,Y 381.346,Z 621.01,A -85,B 0,C 180,E1 -26825.492,E2 -26825.492} C_VEL
LIN {X 0,Y 382.936,Z 625.004,A -85,B 0,C 180,E1 -26828.181,E2 -26828.181} C_VEL
LIN {X 0,Y 383.347,Z 626.204,A -85,B 0,C 180,E1 -26828.758,E2 -26828.758} C_VEL
LIN {X 0,Y 369.395,Z 750.867,A -85,B 0,C 180,E1 -26830.456,E2 -26830.456} C_VEL
LIN {X 0,Y 364.735,Z 776.93,A -85,B 0,C 180,E1 -26830.89,E2 -26830.89} C_VEL
LIN {X 0,Y 359.53,Z 798.316,A -85,B 0,C 180,E1 -26831.346,E2 -26831.346} C_VEL
LIN {X 0,Y 351.715,Z 823.618,A -85,B 0,C 180,E1 -26832.053,E2 -26832.053} C_VEL
LIN {X 0,Y 344.038,Z 843.983,A -85,B 0,C 180,E1 -26832.782,E2 -26832.782} C_VEL
LIN {X 0,Y 334.055,Z 866.593,A -85,B 0,C 180,E1 -26833.783,E2 -26833.783} C_VEL
LIN {X 0,Y 323.806,Z 886.361,A -85,B 0,C 180,E1 -26834.868,E2 -26834.868} C_VEL
LIN {X 0,Y 311.901,Z 906.744,A -85,B 0,C 180,E1 -26836.233,E2 -26836.233} C_VEL
LIN {X 0,Y 298.892,Z 926.11,A -85,B 0,C 180,E1 -26837.873,E2 -26837.873} C_VEL
LIN {X 0,Y 285.72,Z 943.805,A -85,B 0,C 180,E1 -26839.716,E2 -26839.716} C_VEL
LIN {X 0,Y 270.813,Z 961.613,A -85,B 0,C 180,E1 -26842.069,E2 -26842.069} C_VEL
LIN {X 0,Y 257.189,Z 976.435,A -85,B 0,C 180,E1 -26844.532,E2 -26844.532} C_VEL
LIN {X 0,Y 240.969,Z 992.442,A -85,B 0,C 180,E1 -26847.962,E2 -26847.962} C_VEL
LIN {X 0,Y 227.986,Z 1004.221,A -85,B 0,C 180,E1 -26851.216,E2 -26851.216} C_VEL
LIN {X 0,Y 212.436,Z 1017.33,A -85,B 0,C 180,E1 -26855.947,E2 -26855.947} C_VEL
LIN {X 0,Y 200.172,Z 1026.983,A -85,B 0,C 180,E1 -26860.601,E2 -26860.601} C_VEL
LIN {X 0,Y 187.782,Z 1036.411,A -85,B 0,C 180,E1 -26866.616,E2 -26866.616} C_VEL
LIN {X 0,Y 177.487,Z 1043.952,A -85,B 0,C 180,E1 -26873.334,E2 -26873.334} C_VEL
LIN {X 0,Y 169.289,Z 1050.249,A -85,B 0,C 180,E1 -26881.032,E2 -26881.032} C_VEL
LIN {X 0,Y 163.979,Z 1054.539,A -85,B 0,C 180,E1 -26888.915,E2 -26888.915} C_VEL
LIN {X 0,Y 161.252,Z 1057.259,A -85,B 0,C 180,E1 -26896.372,E2 -26896.372} C_VEL
LIN {X 0,Y 160.173,Z 1058.893,A -85,B 0,C 180,E1 -26904.268,E2 -26904.268} C_VEL
LIN {X 0,Y 160.051,Z 1059.182,A -85,B 0,C 180,E1 -26911.074,E2 -26911.074} C_VEL
LIN {X 0,Y 160.322,Z 1058.552,A -85,B 0,C 180,E1 -26917.887,E2 -26917.887} C_VEL
LIN {X 0,Y 161.509,Z 1056.987,A -85,B 0,C 180,E1 -26924.704,E2 -26924.704} C_VEL
LIN {X 0,Y 164.488,Z 1054.153,A -85,B 0,C 180,E1 -26932.141,E2 -26932.141} C_VEL
LIN {X 0,Y 171.018,Z 1048.9,A -85,B 0,C 180,E1 -26940.965,E2 -26940.965} C_VEL
LIN {X 0,Y 178.616,Z 1043.208,A -85,B 0,C 180,E1 -26947.603,E2 -26947.603} C_VEL
LIN {X 0,Y 190.231,Z 1034.653,A -85,B 0,C 180,E1 -26954.798,E2 -26954.798} C_VEL
LIN {X 0,Y 201.822,Z 1025.839,A -85,B 0,C 180,E1 -26960.168,E2 -26960.168} C_VEL
LIN {X 0,Y 216.246,Z 1014.402,A -85,B 0,C 180,E1 -26965.391,E2 -26965.391} C_VEL
LIN {X 0,Y 230.175,Z 1002.469,A -85,B 0,C 180,E1 -26969.452,E2 -26969.452} C_VEL
LIN {X 0,Y 245.479,Z 988.449,A -85,B 0,C 180,E1 -26973.131,E2 -26973.131} C_VEL
LIN {X 0,Y 260.238,Z 973.465,A -85,B 0,C 180,E1 -26976.128,E2 -26976.128} C_VEL
LIN {X 0,Y 275.217,Z 956.954,A -85,B 0,C 180,E1 -26978.732,E2 -26978.732} C_VEL
LIN {X 0,Y 289.408,Z 939.333,A -85,B 0,C 180,E1 -26980.897,E2 -26980.897} C_VEL
LIN {X 0,Y 302.807,Z 921.016,A -85,B 0,C 180,E1 -26982.711,E2 -26982.711} C_VEL
LIN {X 0,Y 315.441,Z 901.313,A -85,B 0,C 180,E1 -26984.268,E2 -26984.268} C_VEL
LIN {X 0,Y 326.381,Z 882.216,A -85,B 0,C 180,E1 -26985.487,E2 -26985.487} C_VEL
LIN {X 0,Y 337.579,Z 859.597,A -85,B 0,C 180,E1 -26986.655,E2 -26986.655} C_VEL
LIN {X 0,Y 345.722,Z 840.54,A -85,B 0,C 180,E1 -26987.452,E2 -26987.452} C_VEL
LIN {X 0,Y 354.377,Z 816.672,A -85,B 0,C 180,E1 -26988.259,E2 -26988.259} C_VEL
LIN {X 0,Y 360.82,Z 794.582,A -85,B 0,C 180,E1 -26988.843,E2 -26988.843} C_VEL
LIN {X 0,Y 366.482,Z 770.141,A -85,B 0,C 180,E1 -26989.339,E2 -26989.339} C_VEL
LIN {X 0,Y 370.308,Z 746.253,A -85,B 0,C 180,E1 -26989.71,E2 -26989.71} C_VEL
LIN {X 0,Y 383.623,Z 626.239,A -85,B 0,C 180,E1 -26991.373,E2 -26991.373} C_VEL
LIN {X 0,Y 382.349,Z 623.197,A -85,B 0,C 180,E1 -26993.242,E2 -26993.242} C_VEL
LIN {X 0,Y 381.324,Z 620.512,A -85,B 0,C 180,E1 -26995.337,E2 -26995.337} C_VEL
LIN {X 0,Y 380.5,Z 617.676,A -85,B 0,C 180,E1 -27000,E2 -27000} C_VEL
LIN {X 0,Y 381.634,Z 621.224,A -85,B 0,C 180,E1 -27005.035,E2 -27005.035} C_VEL
LIN {X 0,Y 383.207,Z 625.148,A -85,B 0,C 180,E1 -27007.723,E2 -27007.723} C_VEL
LIN {X 0,Y 383.686,Z 626.449,A -85,B 0,C 180,E1 -27008.385,E2 -27008.385} C_VEL
LIN {X 0,Y 370.543,Z 745.555,A -85,B 0,C 180,E1 -27010.003,E2 -27010.003} C_VEL
LIN {X 0,Y 369.358,Z 753.223,A -85,B 0,C 180,E1 -27009.954,E2 -27009.954} C_VEL
LIN {X 0,Y 364.653,Z 774.654,A -85,B 0,C 180,E1 -27009.276,E2 -27009.276} C_VEL
LIN {X 0,Y 363.374,Z 780.064,A -85,B 0,C 180,E1 -27009.302,E2 -27009.302} C_VEL
LIN {X 0,Y 357.953,Z 801.918,A -85,B 0,C 180,E1 -27009.699,E2 -27009.699} C_VEL
LIN {X 0,Y 349.896,Z 827.417,A -85,B 0,C 180,E1 -27010.299,E2 -27010.299} C_VEL
LIN {X 0,Y 342.154,Z 847.542,A -85,B 0,C 180,E1 -27010.915,E2 -27010.915} C_VEL
LIN {X 0,Y 331.972,Z 870.225,A -85,B 0,C 180,E1 -27011.793,E2 -27011.793} C_VEL
LIN {X 0,Y 321.472,Z 890.175,A -85,B 0,C 180,E1 -27012.773,E2 -27012.773} C_VEL
LIN {X 0,Y 309.641,Z 910.141,A -85,B 0,C 180,E1 -27013.982,E2 -27013.982} C_VEL
LIN {X 0,Y 296.271,Z 929.836,A -85,B 0,C 180,E1 -27015.483,E2 -27015.483} C_VEL
LIN {X 0,Y 283.503,Z 946.784,A -85,B 0,C 180,E1 -27017.099,E2 -27017.099} C_VEL
LIN {X 0,Y 268.06,Z 965.176,A -85,B 0,C 180,E1 -27019.315,E2 -27019.315} C_VEL
LIN {X 0,Y 253.9,Z 980.401,A -85,B 0,C 180,E1 -27021.658,E2 -27021.658} C_VEL
LIN {X 0,Y 237.867,Z 996.172,A -85,B 0,C 180,E1 -27024.773,E2 -27024.773} C_VEL
LIN {X 0,Y 223.376,Z 1009.142,A -85,B 0,C 180,E1 -27028.136,E2 -27028.136} C_VEL
LIN {X 0,Y 208.382,Z 1021.748,A -85,B 0,C 180,E1 -27032.38,E2 -27032.38} C_VEL
LIN {X 0,Y 194.033,Z 1032.855,A -85,B 0,C 180,E1 -27037.477,E2 -27037.477} C_VEL
LIN {X 0,Y 181.391,Z 1042.367,A -85,B 0,C 180,E1 -27043.312,E2 -27043.312} C_VEL
LIN {X 0,Y 169.877,Z 1050.756,A -85,B 0,C 180,E1 -27050.529,E2 -27050.529} C_VEL
LIN {X 0,Y 161.749,Z 1056.951,A -85,B 0,C 180,E1 -27057.884,E2 -27057.884} C_VEL
LIN {X 0,Y 155.555,Z 1062.181,A -85,B 0,C 180,E1 -27066.914,E2 -27066.914} C_VEL
LIN {X 0,Y 152.915,Z 1065.075,A -85,B 0,C 180,E1 -27074.449,E2 -27074.449} C_VEL
LIN {X 0,Y 152.033,Z 1066.797,A -85,B 0,C 180,E1 -27081.68,E2 -27081.68} C_VEL
LIN {X 0,Y 152.027,Z 1067.46,A -85,B 0,C 180,E1 -27088.115,E2 -27088.115} C_VEL
LIN {X 0,Y 152.004,Z 1067.334,A -85,B 0,C 180,E1 -27093.771,E2 -27093.771} C_VEL
LIN {X 0,Y 152.137,Z 1066.421,A -85,B 0,C 180,E1 -27100.221,E2 -27100.221} C_VEL
LIN {X 0,Y 153.863,Z 1063.961,A -85,B 0,C 180,E1 -27108.961,E2 -27108.961} C_VEL
LIN {X 0,Y 158.114,Z 1059.828,A -85,B 0,C 180,E1 -27117.493,E2 -27117.493} C_VEL
LIN {X 0,Y 164.775,Z 1054.536,A -85,B 0,C 180,E1 -27125.203,E2 -27125.203} C_VEL
LIN {X 0,Y 175.305,Z 1046.679,A -85,B 0,C 180,E1 -27133.192,E2 -27133.192} C_VEL
LIN {X 0,Y 186.328,Z 1038.548,A -85,B 0,C 180,E1 -27139.169,E2 -27139.169} C_VEL
LIN {X 0,Y 201,Z 1027.373,A -85,B 0,C 180,E1 -27145.165,E2 -27145.165} C_VEL
LIN {X 0,Y 214.647,Z 1016.372,A -85,B 0,C 180,E1 -27149.517,E2 -27149.517} C_VEL
LIN {X 0,Y 230.894,Z 1002.355,A -85,B 0,C 180,E1 -27153.69,E2 -27153.69} C_VEL
LIN {X 0,Y 244.979,Z 989.098,A -85,B 0,C 180,E1 -27156.685,E2 -27156.685} C_VEL
LIN {X 0,Y 260.503,Z 973.314,A -85,B 0,C 180,E1 -27159.479,E2 -27159.479} C_VEL
LIN {X 0,Y 274.861,Z 956.998,A -85,B 0,C 180,E1 -27161.707,E2 -27161.707} C_VEL
LIN {X 0,Y 288.289,Z 940.31,A -85,B 0,C 180,E1 -27163.536,E2 -27163.536} C_VEL
LIN {X 0,Y 302.551,Z 920.423,A -85,B 0,C 180,E1 -27165.257,E2 -27165.257} C_VEL
LIN {X 0,Y 314.589,Z 901.568,A -85,B 0,C 180,E1 -27166.553,E2 -27166.553} C_VEL
LIN {X 0,Y 327.351,Z 878.716,A -85,B 0,C 180,E1 -27167.804,E2 -27167.804} C_VEL
LIN {X 0,Y 336.573,Z 859.711,A -85,B 0,C 180,E1 -27168.625,E2 -27168.625} C_VEL
LIN {X 0,Y 346.17,Z 836.875,A -85,B 0,C 180,E1 -27169.414,E2 -27169.414} C_VEL
LIN {X 0,Y 353.576,Z 815.516,A -85,B 0,C 180,E1 -27169.99,E2 -27169.99} C_VEL
LIN {X 0,Y 360.311,Z 792.088,A -85,B 0,C 180,E1 -27170.483,E2 -27170.483} C_VEL
LIN {X 0,Y 365.568,Z 767.431,A -85,B 0,C 180,E1 -27170.892,E2 -27170.892} C_VEL
LIN {X 0,Y 369.112,Z 743.924,A -85,B 0,C 180,E1 -27171.237,E2 -27171.237} C_VEL
LIN {X 0,Y 381.591,Z 632.232,A -85,B 0,C 180,E1 -27172.737,E2 -27172.737} C_VEL
LIN {X 0,Y 380.051,Z 628.28,A -85,B 0,C 180,E1 -27175.624,E2 -27175.624} C_VEL
LIN {X 0,Y 379.231,Z 625.052,A -85,B 0,C 180,E1 -27180.302,E2 -27180.302} C_VEL
LIN {X 0,Y 380.257,Z 628.815,A -85,B 0,C 180,E1 -27185.281,E2 -27185.281} C_VEL
LIN {X 0,Y 381.56,Z 632.213,A -85,B 0,C 180,E1 -27187.646,E2 -27187.646} C_VEL
LIN {X 0,Y 368.027,Z 751.102,A -85,B 0,C 180,E1 -27189.231,E2 -27189.231} C_VEL
LIN {X 0,Y 363.304,Z 777.171,A -85,B 0,C 180,E1 -27189.65,E2 -27189.65} C_VEL
LIN {X 0,Y 357.999,Z 798.692,A -85,B 0,C 180,E1 -27190.092,E2 -27190.092} C_VEL
LIN {X 0,Y 349.874,Z 824.539,A -85,B 0,C 180,E1 -27190.791,E2 -27190.791} C_VEL
LIN {X 0,Y 342.304,Z 844.316,A -85,B 0,C 180,E1 -27191.475,E2 -27191.475} C_VEL
LIN {X 0,Y 332.073,Z 867.117,A -85,B 0,C 180,E1 -27192.448,E2 -27192.448} C_VEL
LIN {X 0,Y 321.829,Z 886.581,A -85,B 0,C 180,E1 -27193.479,E2 -27193.479} C_VEL
LIN {X 0,Y 309.78,Z 906.893,A -85,B 0,C 180,E1 -27194.79,E2 -27194.79} C_VEL
LIN {X 0,Y 296.503,Z 926.331,A -85,B 0,C 180,E1 -27196.38,E2 -27196.38} C_VEL
LIN {X 0,Y 283.081,Z 944.026,A -85,B 0,C 180,E1 -27198.167,E2 -27198.167} C_VEL
LIN {X 0,Y 267.856,Z 961.833,A -85,B 0,C 180,E1 -27200.452,E2 -27200.452} C_VEL
LIN {X 0,Y 253.905,Z 976.656,A -85,B 0,C 180,E1 -27202.854,E2 -27202.854} C_VEL
LIN {X 0,Y 237.343,Z 992.568,A -85,B 0,C 180,E1 -27206.19,E2 -27206.19} C_VEL
LIN {X 0,Y 223.748,Z 1004.524,A -85,B 0,C 180,E1 -27209.444,E2 -27209.444} C_VEL
LIN {X 0,Y 207.719,Z 1017.551,A -85,B 0,C 180,E1 -27214.112,E2 -27214.112} C_VEL
LIN {X 0,Y 194.92,Z 1027.203,A -85,B 0,C 180,E1 -27218.766,E2 -27218.766} C_VEL
LIN {X 0,Y 181.895,Z 1036.632,A -85,B 0,C 180,E1 -27224.837,E2 -27224.837} C_VEL
LIN {X 0,Y 170.972,Z 1044.172,A -85,B 0,C 180,E1 -27231.69,E2 -27231.69} C_VEL
LIN {X 0,Y 162.099,Z 1050.521,A -85,B 0,C 180,E1 -27239.721,E2 -27239.721} C_VEL
LIN {X 0,Y 156.22,Z 1054.911,A -85,B 0,C 180,E1 -27248.209,E2 -27248.209} C_VEL
LIN {X 0,Y 153.309,Z 1057.585,A -85,B 0,C 180,E1 -27256.036,E2 -27256.036} C_VEL
LIN {X 0,Y 152.171,Z 1059.128,A -85,B 0,C 180,E1 -27264.344,E2 -27264.344} C_VEL
LIN {X 0,Y 152.054,Z 1059.395,A -85,B 0,C 180,E1 -27271.131,E2 -27271.131} C_VEL
LIN {X 0,Y 152.362,Z 1058.766,A -85,B 0,C 180,E1 -27278.302,E2 -27278.302} C_VEL
LIN {X 0,Y 153.781,Z 1057.112,A -85,B 0,C 180,E1 -27285.781,E2 -27285.781} C_VEL
LIN {X 0,Y 157.396,Z 1054.062,A -85,B 0,C 180,E1 -27293.99,E2 -27293.99} C_VEL
LIN {X 0,Y 164.388,Z 1048.87,A -85,B 0,C 180,E1 -27302.775,E2 -27302.775} C_VEL
LIN {X 0,Y 172.721,Z 1043.063,A -85,B 0,C 180,E1 -27309.651,E2 -27309.651} C_VEL
LIN {X 0,Y 184.999,Z 1034.494,A -85,B 0,C 180,E1 -27316.858,E2 -27316.858} C_VEL
LIN {X 0,Y 196.798,Z 1025.953,A -85,B 0,C 180,E1 -27322.064,E2 -27322.064} C_VEL
LIN {X 0,Y 211.686,Z 1014.619,A -85,B 0,C 180,E1 -27327.222,E2 -27327.222} C_VEL
LIN {X 0,Y 225.931,Z 1002.843,A -85,B 0,C 180,E1 -27331.197,E2 -27331.197} C_VEL
LIN {X 0,Y 241.285,Z 989.25,A -85,B 0,C 180,E1 -27334.733,E2 -27334.733} C_VEL
LIN {X 0,Y 256.227,Z 974.517,A -85,B 0,C 180,E1 -27337.647,E2 -27337.647} C_VEL
LIN {X 0,Y 270.263,Z 959.483,A -85,B 0,C 180,E1 -27340.005,E2 -27340.005} C_VEL
LIN {X 0,Y 285.685,Z 941.036,A -85,B 0,C 180,E1 -27342.272,E2 -27342.272} C_VEL
LIN {X 0,Y 298.598,Z 923.835,A -85,B 0,C 180,E1 -27343.957,E2 -27343.957} C_VEL
LIN {X 0,Y 312.758,Z 902.485,A -85,B 0,C 180,E1 -27345.626,E2 -27345.626} C_VEL
LIN {X 0,Y 323.646,Z 883.867,A -85,B 0,C 180,E1 -27346.784,E2 -27346.784} C_VEL
LIN {X 0,Y 335.438,Z 860.626,A -85,B 0,C 180,E1 -27347.956,E2 -27347.956} C_VEL
LIN {X 0,Y 344.066,Z 840.747,A -85,B 0,C 180,E1 -27348.758,E2 -27348.758} C_VEL
LIN {X 0,Y 352.832,Z 816.877,A -85,B 0,C 180,E1 -27349.534,E2 -27349.534} C_VEL
LIN {X 0,Y 359.353,Z 794.792,A -85,B 0,C 180,E1 -27350.097,E2 -27350.097} C_VEL
LIN {X 0,Y 365.099,Z 770.26,A -85,B 0,C 180,E1 -27350.576,E2 -27350.576} C_VEL
LIN {X 0,Y 368.962,Z 746.445,A -85,B 0,C 180,E1 -27350.933,E2 -27350.933} C_VEL
LIN {X 0,Y 381.832,Z 632.426,A -85,B 0,C 180,E1 -27352.476,E2 -27352.476} C_VEL
LIN {X 0,Y 380.282,Z 628.396,A -85,B 0,C 180,E1 -27355.476,E2 -27355.476} C_VEL
LIN {X 0,Y 379.52,Z 625.653,A -85,B 0,C 180,E1 -27360,E2 -27360} C_VEL
LIN {X 0,Y 380.546,Z 629.026,A -85,B 0,C 180,E1 -27364.823,E2 -27364.823} C_VEL
LIN {X 0,Y 381.892,Z 632.528,A -85,B 0,C 180,E1 -27367.277,E2 -27367.277} C_VEL
LIN {X 0,Y 368.059,Z 754.17,A -85,B 0,C 180,E1 -27368.9,E2 -27368.9} C_VEL
LIN {X 0,Y 363.374,Z 780.064,A -85,B 0,C 180,E1 -27369.302,E2 -27369.302} C_VEL
LIN {X 0,Y 361.51,Z 787.588,A -85,B 0,C 180,E1 -27369.258,E2 -27369.258} C_VEL
LIN {X 0,Y 355.184,Z 807.498,A -85,B 0,C 180,E1 -27368.649,E2 -27368.649} C_VEL
LIN {X 0,Y 353.055,Z 813.807,A -85,B 0,C 180,E1 -27368.68,E2 -27368.68} C_VEL
LIN {X 0,Y 345.908,Z 834.412,A -85,B 0,C 180,E1 -27369.195,E2 -27369.195} C_VEL
LIN {X 0,Y 336.023,Z 858.095,A -85,B 0,C 180,E1 -27369.954,E2 -27369.954} C_VEL
LIN {X 0,Y 326.16,Z 878.256,A -85,B 0,C 180,E1 -27370.778,E2 -27370.778} C_VEL
LIN {X 0,Y 313.142,Z 901.28,A -85,B 0,C 180,E1 -27371.979,E2 -27371.979} C_VEL
LIN {X 0,Y 301.392,Z 919.438,A -85,B 0,C 180,E1 -27373.167,E2 -27373.167} C_VEL
LIN {X 0,Y 286.988,Z 939.305,A -85,B 0,C 180,E1 -27374.797,E2 -27374.797} C_VEL
LIN {X 0,Y 273.288,Z 956.054,A -85,B 0,C 180,E1 -27376.546,E2 -27376.546} C_VEL
LIN {X 0,Y 258.17,Z 972.902,A -85,B 0,C 180,E1 -27378.751,E2 -27378.751} C_VEL
LIN {X 0,Y 241.849,Z 989.097,A -85,B 0,C 180,E1 -27381.529,E2 -27381.529} C_VEL
LIN {X 0,Y 226.581,Z 1003.037,A -85,B 0,C 180,E1 -27384.623,E2 -27384.623} C_VEL
LIN {X 0,Y 210.579,Z 1016.304,A -85,B 0,C 180,E1 -27388.546,E2 -27388.546} C_VEL
LIN {X 0,Y 196.391,Z 1027.285,A -85,B 0,C 180,E1 -27392.852,E2 -27392.852} C_VEL
LIN {X 0,Y 181.023,Z 1038.433,A -85,B 0,C 180,E1 -27398.847,E2 -27398.847} C_VEL
LIN {X 0,Y 169.361,Z 1046.552,A -85,B 0,C 180,E1 -27404.889,E2 -27404.889} C_VEL
LIN {X 0,Y 157.704,Z 1054.641,A -85,B 0,C 180,E1 -27413.417,E2 -27413.417} C_VEL
LIN {X 0,Y 150.858,Z 1059.66,A -85,B 0,C 180,E1 -27421.063,E2 -27421.063} C_VEL
LIN {X 0,Y 146.016,Z 1063.906,A -85,B 0,C 180,E1 -27430.394,E2 -27430.394} C_VEL
LIN {X 0,Y 144.18,Z 1066.222,A -85,B 0,C 180,E1 -27439.208,E2 -27439.208} C_VEL
LIN {X 0,Y 144.004,Z 1067.126,A -85,B 0,C 180,E1 -27446.018,E2 -27446.018} C_VEL
LIN {X 0,Y 144.032,Z 1067.265,A -85,B 0,C 180,E1 -27451.591,E2 -27451.591} C_VEL
LIN {X 0,Y 144.035,Z 1066.637,A -85,B 0,C 180,E1 -27458.382,E2 -27458.382} C_VEL
LIN {X 0,Y 144.988,Z 1064.948,A -85,B 0,C 180,E1 -27466.013,E2 -27466.013} C_VEL
LIN {X 0,Y 147.953,Z 1061.991,A -85,B 0,C 180,E1 -27474.166,E2 -27474.166} C_VEL
LIN {X 0,Y 154.813,Z 1056.667,A -85,B 0,C 180,E1 -27483.741,E2 -27483.741} C_VEL
LIN {X 0,Y 163.562,Z 1050.456,A -85,B 0,C 180,E1 -27491.317,E2 -27491.317} C_VEL
LIN {X 0,Y 175.793,Z 1042.038,A -85,B 0,C 180,E1 -27498.659,E2 -27498.659} C_VEL
LIN {X 0,Y 189.09,Z 1032.514,A -85,B 0,C 180,E1 -27504.521,E2 -27504.521} C_VEL
LIN {X 0,Y 204.05,Z 1021.381,A -85,B 0,C 180,E1 -27509.591,E2 -27509.591} C_VEL
LIN {X 0,Y 219.692,Z 1008.654,A -85,B 0,C 180,E1 -27513.802,E2 -27513.802} C_VEL
LIN {X 0,Y 236.129,Z 994.321,A -85,B 0,C 180,E1 -27517.386,E2 -27517.386} C_VEL
LIN {X 0,Y 251.804,Z 979.086,A -85,B 0,C 180,E1 -27520.238,E2 -27520.238} C_VEL
LIN {X 0,Y 267.177,Z 962.822,A -85,B 0,C 180,E1 -27522.615,E2 -27522.615} C_VEL
LIN {X 0,Y 282.518,Z 944.56,A -85,B 0,C 180,E1 -27524.672,E2 -27524.672} C_VEL
LIN {X 0,Y 295.941,Z 926.862,A -85,B 0,C 180,E1 -27526.256,E2 -27526.256} C_VEL
LIN {X 0,Y 309.688,Z 906.354,A -85,B 0,C 180,E1 -27527.696,E2 -27527.696} C_VEL
LIN {X 0,Y 321.101,Z 887.094,A -85,B 0,C 180,E1 -27528.78,E2 -27528.78} C_VEL
LIN {X 0,Y 333.203,Z 863.523,A -85,B 0,C 180,E1 -27529.826,E2 -27529.826} C_VEL
LIN {X 0,Y 341.649,Z 844.359,A -85,B 0,C 180,E1 -27530.499,E2 -27530.499} C_VEL
LIN {X 0,Y 350.622,Z 820.432,A -85,B 0,C 180,E1 -27531.164,E2 -27531.164} C_VEL
LIN {X 0,Y 357.417,Z 797.892,A -85,B 0,C 180,E1 -27531.638,E2 -27531.638} C_VEL
LIN {X 0,Y 363.265,Z 773.383,A -85,B 0,C 180,E1 -27532.048,E2 -27532.048} C_VEL
LIN {X 0,Y 367.204,Z 749.376,A -85,B 0,C 180,E1 -27532.395,E2 -27532.395} C_VEL
LIN {X 0,Y 379.9,Z 638.685,A -85,B 0,C 180,E1 -27533.843,E2 -27533.843} C_VEL
LIN {X 0,Y 378.943,Z 636.064,A -85,B 0,C 180,E1 -27535.915,E2 -27535.915} C_VEL
LIN {X 0,Y 378.249,Z 633.051,A -85,B 0,C 180,E1 -27540.303,E2 -27540.303} C_VEL
LIN {X 0,Y 379.201,Z 636.732,A -85,B 0,C 180,E1 -27545.144,E2 -27545.144} C_VEL
LIN {X 0,Y 379.85,Z 638.842,A -85,B 0,C 180,E1 -27546.535,E2 -27546.535} C_VEL
LIN {X 0,Y 366.814,Z 751.449,A -85,B 0,C 180,E1 -27547.999,E2 -27547.999} C_VEL
LIN {X 0,Y 362.045,Z 777.409,A -85,B 0,C 180,E1 -27548.401,E2 -27548.401} C_VEL
LIN {X 0,Y 356.682,Z 798.916,A -85,B 0,C 180,E1 -27548.824,E2 -27548.824} C_VEL
LIN {X 0,Y 348.717,Z 824.062,A -85,B 0,C 180,E1 -27549.473,E2 -27549.473} C_VEL
LIN {X 0,Y 340.796,Z 844.538,A -85,B 0,C 180,E1 -27550.15,E2 -27550.15} C_VEL
LIN {X 0,Y 330.613,Z 866.984,A -85,B 0,C 180,E1 -27551.068,E2 -27551.068} C_VEL
LIN {X 0,Y 319.895,Z 887.065,A -85,B 0,C 180,E1 -27552.088,E2 -27552.088} C_VEL
LIN {X 0,Y 307.317,Z 907.877,A -85,B 0,C 180,E1 -27553.388,E2 -27553.388} C_VEL
LIN {X 0,Y 293.873,Z 927.156,A -85,B 0,C 180,E1 -27554.919,E2 -27554.919} C_VEL
LIN {X 0,Y 279.346,Z 945.885,A -85,B 0,C 180,E1 -27556.767,E2 -27556.767} C_VEL
